LIN {X 0,Y 474.608,Z 139.367,A -85,B 0,C 180,E1 -7425.895,E2 -7425.895} C_VEL
LIN {X 0,Y 474.709,Z 139.486,A -85,B 0,C 180,E1 -7429.16,E2 -7429.16} C_VEL
LIN {X 0,Y 475.786,Z 146.089,A -85,B 0,C 180,E1 -7430.567,E2 -7430.567} C_VEL
LIN {X 0,Y 475.59,Z 156.694,A -85,B 0,C 180,E1 -7432.708,E2 -7432.708} C_VEL
LIN {X 0,Y 475.534,Z 159.268,A -85,B 0,C 180,E1 -7433.227,E2 -7433.227} C_VEL
LIN {X 0,Y 478.307,Z 173.098,A -85,B 0,C 180,E1 -7433.565,E2 -7433.565} C_VEL
LIN {X 0,Y 477.544,Z 266.711,A -85,B 0,C 180,E1 -7435.018,E2 -7435.018} C_VEL
LIN {X 0,Y 477.306,Z 280.071,A -85,B 0,C 180,E1 -7435.404,E2 -7435.404} C_VEL
LIN {X 0,Y 477.288,Z 280.718,A -85,B 0,C 180,E1 -7435.427,E2 -7435.427} C_VEL
LIN {X 0,Y 476.628,Z 286.343,A -85,B 0,C 180,E1 -7435.627,E2 -7435.627} C_VEL
LIN {X 0,Y 473.579,Z 295.359,A -85,B 0,C 180,E1 -7435.964,E2 -7435.964} C_VEL
LIN {X 0,Y 470.344,Z 304.06,A -85,B 0,C 180,E1 -7436.39,E2 -7436.39} C_VEL
LIN {X 0,Y 469.403,Z 309.194,A -85,B 0,C 180,E1 -7436.728,E2 -7436.728} C_VEL
LIN {X 0,Y 468.945,Z 319.732,A -85,B 0,C 180,E1 -7437.603,E2 -7437.603} C_VEL
LIN {X 0,Y 468.482,Z 329.529,A -85,B 0,C 180,E1 -7438.608,E2 -7438.608} C_VEL
LIN {X 0,Y 467.98,Z 338.944,A -85,B 0,C 180,E1 -7439.795,E2 -7439.795} C_VEL
LIN {X 0,Y 467.628,Z 346.312,A -85,B 0,C 180,E1 -7440.941,E2 -7440.941} C_VEL
LIN {X 0,Y 467.263,Z 352.96,A -85,B 0,C 180,E1 -7442.208,E2 -7442.208} C_VEL
LIN {X 0,Y 467.028,Z 358.937,A -85,B 0,C 180,E1 -7443.645,E2 -7443.645} C_VEL
LIN {X 0,Y 466.831,Z 363.471,A -85,B 0,C 180,E1 -7445.069,E2 -7445.069} C_VEL
LIN {X 0,Y 466.694,Z 367.163,A -85,B 0,C 180,E1 -7446.722,E2 -7446.722} C_VEL
LIN {X 0,Y 466.58,Z 368.845,A -85,B 0,C 180,E1 -7447.879,E2 -7447.879} C_VEL
LIN {X 0,Y 466.563,Z 369.776,A -85,B 0,C 180,E1 -7449.054,E2 -7449.054} C_VEL
LIN {X 0,Y 466.57,Z 369.919,A -85,B 0,C 180,E1 -7450.647,E2 -7450.647} C_VEL
LIN {X 0,Y 466.589,Z 369.328,A -85,B 0,C 180,E1 -7451.609,E2 -7451.609} C_VEL
LIN {X 0,Y 466.604,Z 368.392,A -85,B 0,C 180,E1 -7452.468,E2 -7452.468} C_VEL
LIN {X 0,Y 466.676,Z 366.991,A -85,B 0,C 180,E1 -7453.373,E2 -7453.373} C_VEL
LIN {X 0,Y 466.797,Z 364.598,A -85,B 0,C 180,E1 -7454.485,E2 -7454.485} C_VEL
LIN {X 0,Y 466.946,Z 359.956,A -85,B 0,C 180,E1 -7456.065,E2 -7456.065} C_VEL
LIN {X 0,Y 467.236,Z 353.669,A -85,B 0,C 180,E1 -7457.623,E2 -7457.623} C_VEL
LIN {X 0,Y 467.517,Z 346.823,A -85,B 0,C 180,E1 -7458.95,E2 -7458.95} C_VEL
LIN {X 0,Y 467.878,Z 338.315,A -85,B 0,C 180,E1 -7460.271,E2 -7460.271} C_VEL
LIN {X 0,Y 468.347,Z 329.513,A -85,B 0,C 180,E1 -7461.37,E2 -7461.37} C_VEL
LIN {X 0,Y 468.844,Z 318.706,A -85,B 0,C 180,E1 -7462.463,E2 -7462.463} C_VEL
LIN {X 0,Y 469.333,Z 307.899,A -85,B 0,C 180,E1 -7463.336,E2 -7463.336} C_VEL
LIN {X 0,Y 469.76,Z 295.801,A -85,B 0,C 180,E1 -7464.096,E2 -7464.096} C_VEL
LIN {X 0,Y 470.119,Z 283.179,A -85,B 0,C 180,E1 -7464.693,E2 -7464.693} C_VEL
LIN {X 0,Y 470.413,Z 270.759,A -85,B 0,C 180,E1 -7465.099,E2 -7465.099} C_VEL
LIN {X 0,Y 470.555,Z 255.199,A -85,B 0,C 180,E1 -7465.396,E2 -7465.396} C_VEL
LIN {X 0,Y 471.161,Z 173.344,A -85,B 0,C 180,E1 -7466.66,E2 -7466.66} C_VEL
LIN {X 0,Y 468.382,Z 159.359,A -85,B 0,C 180,E1 -7466.99,E2 -7466.99} C_VEL
LIN {X 0,Y 468.71,Z 147.809,A -85,B 0,C 180,E1 -7469.356,E2 -7469.356} C_VEL
LIN {X 0,Y 468.548,Z 144.722,A -85,B 0,C 180,E1 -7470,E2 -7470} C_VEL
LIN {X 0,Y 467.639,Z 140.235,A -85,B 0,C 180,E1 -7471.023,E2 -7471.023} C_VEL
LIN {X 0,Y 467.806,Z 140.215,A -85,B 0,C 180,E1 -7472.583,E2 -7472.583} C_VEL
LIN {X 0,Y 467.695,Z 140.229,A -85,B 0,C 180,E1 -7476.038,E2 -7476.038} C_VEL
LIN {X 0,Y 467.628,Z 140.231,A -85,B 0,C 180,E1 -7478.644,E2 -7478.644} C_VEL
LIN {X 0,Y 467.643,Z 140.232,A -85,B 0,C 180,E1 -7482.146,E2 -7482.146} C_VEL
LIN {X 0,Y 467.572,Z 140.246,A -85,B 0,C 180,E1 -7485.698,E2 -7485.698} C_VEL
LIN {X 0,Y 467.564,Z 140.239,A -85,B 0,C 180,E1 -7488.747,E2 -7488.747} C_VEL
LIN {X 0,Y 467.51,Z 140.247,A -85,B 0,C 180,E1 -7492.075,E2 -7492.075} C_VEL
LIN {X 0,Y 467.523,Z 140.245,A -85,B 0,C 180,E1 -7494.892,E2 -7494.892} C_VEL
LIN {X 0,Y 467.533,Z 140.246,A -85,B 0,C 180,E1 -7497.775,E2 -7497.775} C_VEL
LIN {X 0,Y 467.524,Z 140.248,A -85,B 0,C 180,E1 -7501.037,E2 -7501.037} C_VEL
LIN {X 0,Y 467.56,Z 140.239,A -85,B 0,C 180,E1 -7504.238,E2 -7504.238} C_VEL
LIN {X 0,Y 467.511,Z 140.253,A -85,B 0,C 180,E1 -7507.181,E2 -7507.181} C_VEL
LIN {X 0,Y 467.538,Z 140.242,A -85,B 0,C 180,E1 -7510.269,E2 -7510.269} C_VEL
LIN {X 0,Y 467.515,Z 140.247,A -85,B 0,C 180,E1 -7512.569,E2 -7512.569} C_VEL
LIN {X 0,Y 467.561,Z 140.246,A -85,B 0,C 180,E1 -7515.053,E2 -7515.053} C_VEL
LIN {X 0,Y 467.559,Z 140.246,A -85,B 0,C 180,E1 -7518.727,E2 -7518.727} C_VEL
LIN {X 0,Y 467.54,Z 140.242,A -85,B 0,C 180,E1 -7521.954,E2 -7521.954} C_VEL
LIN {X 0,Y 467.545,Z 140.243,A -85,B 0,C 180,E1 -7525.166,E2 -7525.166} C_VEL
LIN {X 0,Y 467.543,Z 140.245,A -85,B 0,C 180,E1 -7528.257,E2 -7528.257} C_VEL
LIN {X 0,Y 467.525,Z 140.244,A -85,B 0,C 180,E1 -7531.248,E2 -7531.248} C_VEL
LIN {X 0,Y 467.563,Z 140.246,A -85,B 0,C 180,E1 -7534.406,E2 -7534.406} C_VEL
LIN {X 0,Y 467.551,Z 140.242,A -85,B 0,C 180,E1 -7536.995,E2 -7536.995} C_VEL
LIN {X 0,Y 467.54,Z 140.243,A -85,B 0,C 180,E1 -7539.774,E2 -7539.774} C_VEL
LIN {X 0,Y 467.554,Z 140.245,A -85,B 0,C 180,E1 -7542.505,E2 -7542.505} C_VEL
LIN {X 0,Y 467.564,Z 140.239,A -85,B 0,C 180,E1 -7545.196,E2 -7545.196} C_VEL
LIN {X 0,Y 467.652,Z 140.232,A -85,B 0,C 180,E1 -7547.855,E2 -7547.855} C_VEL
LIN {X 0,Y 467.633,Z 140.231,A -85,B 0,C 180,E1 -7551.357,E2 -7551.357} C_VEL
LIN {X 0,Y 467.704,Z 140.229,A -85,B 0,C 180,E1 -7553.963,E2 -7553.963} C_VEL
LIN {X 0,Y 467.815,Z 140.21,A -85,B 0,C 180,E1 -7557.417,E2 -7557.417} C_VEL
LIN {X 0,Y 467.853,Z 140.208,A -85,B 0,C 180,E1 -7560,E2 -7560} C_VEL
LIN {X 0,Y 467.815,Z 140.208,A -85,B 0,C 180,E1 -7562.584,E2 -7562.584} C_VEL
LIN {X 0,Y 467.698,Z 140.225,A -85,B 0,C 180,E1 -7566.038,E2 -7566.038} C_VEL
LIN {X 0,Y 467.64,Z 140.229,A -85,B 0,C 180,E1 -7568.644,E2 -7568.644} C_VEL
LIN {X 0,Y 467.662,Z 140.228,A -85,B 0,C 180,E1 -7572.146,E2 -7572.146} C_VEL
LIN {X 0,Y 467.618,Z 140.237,A -85,B 0,C 180,E1 -7575.696,E2 -7575.696} C_VEL
LIN {X 0,Y 467.62,Z 140.239,A -85,B 0,C 180,E1 -7579.308,E2 -7579.308} C_VEL
LIN {X 0,Y 467.529,Z 140.243,A -85,B 0,C 180,E1 -7582.075,E2 -7582.075} C_VEL
LIN {X 0,Y 467.56,Z 140.243,A -85,B 0,C 180,E1 -7584.89,E2 -7584.89} C_VEL
LIN {X 0,Y 467.548,Z 140.242,A -85,B 0,C 180,E1 -7587.774,E2 -7587.774} C_VEL
LIN {X 0,Y 467.542,Z 140.249,A -85,B 0,C 180,E1 -7591.038,E2 -7591.038} C_VEL
LIN {X 0,Y 467.581,Z 140.237,A -85,B 0,C 180,E1 -7594.24,E2 -7594.24} C_VEL
LIN {X 0,Y 467.547,Z 140.245,A -85,B 0,C 180,E1 -7597.185,E2 -7597.185} C_VEL
LIN {X 0,Y 467.562,Z 140.241,A -85,B 0,C 180,E1 -7600.267,E2 -7600.267} C_VEL
LIN {X 0,Y 467.549,Z 140.241,A -85,B 0,C 180,E1 -7603.746,E2 -7603.746} C_VEL
LIN {X 0,Y 467.549,Z 140.243,A -85,B 0,C 180,E1 -7606.254,E2 -7606.254} C_VEL
LIN {X 0,Y 467.561,Z 140.239,A -85,B 0,C 180,E1 -7609.733,E2 -7609.733} C_VEL
LIN {X 0,Y 467.546,Z 140.245,A -85,B 0,C 180,E1 -7612.815,E2 -7612.815} C_VEL
LIN {X 0,Y 467.58,Z 140.238,A -85,B 0,C 180,E1 -7615.76,E2 -7615.76} C_VEL
LIN {X 0,Y 467.569,Z 140.242,A -85,B 0,C 180,E1 -7618.956,E2 -7618.956} C_VEL
LIN {X 0,Y 467.549,Z 140.25,A -85,B 0,C 180,E1 -7622.226,E2 -7622.226} C_VEL
LIN {X 0,Y 467.586,Z 140.323,A -85,B 0,C 180,E1 -7624.069,E2 -7624.069} C_VEL
LIN {X 0,Y 469.75,Z 151.558,A -85,B 0,C 180,E1 -7626.174,E2 -7626.174} C_VEL
LIN {X 0,Y 469.254,Z 166.324,A -85,B 0,C 180,E1 -7628.746,E2 -7628.746} C_VEL
LIN {X 0,Y 468.414,Z 185.761,A -85,B 0,C 180,E1 -7632.086,E2 -7632.086} C_VEL
LIN {X 0,Y 468.271,Z 191.496,A -85,B 0,C 180,E1 -7633.045,E2 -7633.045} C_VEL
LIN {X 0,Y 471.064,Z 211.651,A -85,B 0,C 180,E1 -7633.456,E2 -7633.456} C_VEL
LIN {X 0,Y 470.402,Z 300.211,A -85,B 0,C 180,E1 -7634.843,E2 -7634.843} C_VEL
LIN {X 0,Y 470.047,Z 313.325,A -85,B 0,C 180,E1 -7635.219,E2 -7635.219} C_VEL
LIN {X 0,Y 469.617,Z 324.856,A -85,B 0,C 180,E1 -7635.704,E2 -7635.704} C_VEL
LIN {X 0,Y 469.114,Z 336.418,A -85,B 0,C 180,E1 -7636.352,E2 -7636.352} C_VEL
LIN {X 0,Y 468.642,Z 348.04,A -85,B 0,C 180,E1 -7637.201,E2 -7637.201} C_VEL
LIN {X 0,Y 468.175,Z 358.889,A -85,B 0,C 180,E1 -7638.198,E2 -7638.198} C_VEL
LIN {X 0,Y 467.738,Z 367.56,A -85,B 0,C 180,E1 -7639.174,E2 -7639.174} C_VEL
LIN {X 0,Y 467.413,Z 375.553,A -85,B 0,C 180,E1 -7640.261,E2 -7640.261} C_VEL
LIN {X 0,Y 467.087,Z 383.366,A -85,B 0,C 180,E1 -7641.564,E2 -7641.564} C_VEL
LIN {X 0,Y 466.831,Z 390.534,A -85,B 0,C 180,E1 -7643.082,E2 -7643.082} C_VEL
LIN {X 0,Y 466.73,Z 395.31,A -85,B 0,C 180,E1 -7644.383,E2 -7644.383} C_VEL
LIN {X 0,Y 466.646,Z 398.958,A -85,B 0,C 180,E1 -7645.681,E2 -7645.681} C_VEL
LIN {X 0,Y 466.69,Z 400.845,A -85,B 0,C 180,E1 -7646.546,E2 -7646.546} C_VEL
LIN {X 0,Y 466.662,Z 402.259,A -85,B 0,C 180,E1 -7647.41,E2 -7647.41} C_VEL
LIN {X 0,Y 466.623,Z 403.879,A -85,B 0,C 180,E1 -7649.137,E2 -7649.137} C_VEL
LIN {X 0,Y 466.605,Z 404.104,A -85,B 0,C 180,E1 -7650,E2 -7650} C_VEL
LIN {X 0,Y 466.623,Z 403.896,A -85,B 0,C 180,E1 -7650.863,E2 -7650.863} C_VEL
LIN {X 0,Y 466.662,Z 402.295,A -85,B 0,C 180,E1 -7652.589,E2 -7652.589} C_VEL
LIN {X 0,Y 466.689,Z 400.901,A -85,B 0,C 180,E1 -7653.453,E2 -7653.453} C_VEL
LIN {X 0,Y 466.687,Z 397.963,A -85,B 0,C 180,E1 -7654.751,E2 -7654.751} C_VEL
LIN {X 0,Y 466.725,Z 393.99,A -85,B 0,C 180,E1 -7656.05,E2 -7656.05} C_VEL
LIN {X 0,Y 466.938,Z 387.896,A -85,B 0,C 180,E1 -7657.568,E2 -7657.568} C_VEL
LIN {X 0,Y 467.178,Z 381.231,A -85,B 0,C 180,E1 -7658.87,E2 -7658.87} C_VEL
LIN {X 0,Y 467.5,Z 372.967,A -85,B 0,C 180,E1 -7660.174,E2 -7660.174} C_VEL
LIN {X 0,Y 467.977,Z 364.522,A -85,B 0,C 180,E1 -7661.258,E2 -7661.258} C_VEL
LIN {X 0,Y 468.416,Z 354.6,A -85,B 0,C 180,E1 -7662.299,E2 -7662.299} C_VEL
LIN {X 0,Y 468.902,Z 343.815,A -85,B 0,C 180,E1 -7663.213,E2 -7663.213} C_VEL
LIN {X 0,Y 469.449,Z 332.569,A -85,B 0,C 180,E1 -7663.969,E2 -7663.969} C_VEL
LIN {X 0,Y 469.961,Z 321.173,A -85,B 0,C 180,E1 -7664.562,E2 -7664.562} C_VEL
LIN {X 0,Y 470.38,Z 308.209,A -85,B 0,C 180,E1 -7665.046,E2 -7665.046} C_VEL
LIN {X 0,Y 470.76,Z 294.419,A -85,B 0,C 180,E1 -7665.366,E2 -7665.366} C_VEL
LIN {X 0,Y 471.211,Z 209.62,A -85,B 0,C 180,E1 -7666.69,E2 -7666.69} C_VEL
LIN {X 0,Y 468.299,Z 190.956,A -85,B 0,C 180,E1 -7667.111,E2 -7667.111} C_VEL
LIN {X 0,Y 468.996,Z 173.231,A -85,B 0,C 180,E1 -7670.161,E2 -7670.161} C_VEL
LIN {X 0,Y 469.879,Z 154.997,A -85,B 0,C 180,E1 -7673.351,E2 -7673.351} C_VEL
LIN {X 0,Y 469.707,Z 150.782,A -85,B 0,C 180,E1 -7674.116,E2 -7674.116} C_VEL
LIN {X 0,Y 467.582,Z 140.244,A -85,B 0,C 180,E1 -7676.171,E2 -7676.171} C_VEL
LIN {X 0,Y 467.553,Z 140.251,A -85,B 0,C 180,E1 -7679.328,E2 -7679.328} C_VEL
LIN {X 0,Y 467.58,Z 140.242,A -85,B 0,C 180,E1 -7681.74,E2 -7681.74} C_VEL
LIN {X 0,Y 467.556,Z 140.239,A -85,B 0,C 180,E1 -7684.833,E2 -7684.833} C_VEL
LIN {X 0,Y 467.554,Z 140.243,A -85,B 0,C 180,E1 -7688.046,E2 -7688.046} C_VEL
LIN {X 0,Y 467.562,Z 140.241,A -85,B 0,C 180,E1 -7691.274,E2 -7691.274} C_VEL
LIN {X 0,Y 467.566,Z 140.244,A -85,B 0,C 180,E1 -7694.948,E2 -7694.948} C_VEL
LIN {X 0,Y 467.556,Z 140.244,A -85,B 0,C 180,E1 -7698.594,E2 -7698.594} C_VEL
LIN {X 0,Y 467.537,Z 140.241,A -85,B 0,C 180,E1 -7701.952,E2 -7701.952} C_VEL
LIN {X 0,Y 467.54,Z 140.243,A -85,B 0,C 180,E1 -7705.165,E2 -7705.165} C_VEL
LIN {X 0,Y 467.544,Z 140.245,A -85,B 0,C 180,E1 -7708.257,E2 -7708.257} C_VEL
LIN {X 0,Y 467.527,Z 140.244,A -85,B 0,C 180,E1 -7711.247,E2 -7711.247} C_VEL
LIN {X 0,Y 467.564,Z 140.242,A -85,B 0,C 180,E1 -7714.405,E2 -7714.405} C_VEL
LIN {X 0,Y 467.552,Z 140.237,A -85,B 0,C 180,E1 -7716.994,E2 -7716.994} C_VEL
LIN {X 0,Y 467.537,Z 140.244,A -85,B 0,C 180,E1 -7719.773,E2 -7719.773} C_VEL
LIN {X 0,Y 467.555,Z 140.243,A -85,B 0,C 180,E1 -7722.504,E2 -7722.504} C_VEL
LIN {X 0,Y 467.592,Z 140.236,A -85,B 0,C 180,E1 -7725.196,E2 -7725.196} C_VEL
LIN {X 0,Y 467.651,Z 140.228,A -85,B 0,C 180,E1 -7727.854,E2 -7727.854} C_VEL
LIN {X 0,Y 467.658,Z 140.226,A -85,B 0,C 180,E1 -7731.356,E2 -7731.356} C_VEL
LIN {X 0,Y 467.706,Z 140.227,A -85,B 0,C 180,E1 -7733.962,E2 -7733.962} C_VEL
LIN {X 0,Y 467.816,Z 140.205,A -85,B 0,C 180,E1 -7737.416,E2 -7737.416} C_VEL
LIN {X 0,Y 467.855,Z 140.203,A -85,B 0,C 180,E1 -7740,E2 -7740} C_VEL
LIN {X 0,Y 467.852,Z 140.202,A -85,B 0,C 180,E1 -7742.582,E2 -7742.582} C_VEL
LIN {X 0,Y 467.715,Z 140.218,A -85,B 0,C 180,E1 -7746.037,E2 -7746.037} C_VEL
LIN {X 0,Y 467.669,Z 140.227,A -85,B 0,C 180,E1 -7748.642,E2 -7748.642} C_VEL
LIN {X 0,Y 467.658,Z 140.228,A -85,B 0,C 180,E1 -7752.145,E2 -7752.145} C_VEL
LIN {X 0,Y 467.64,Z 140.232,A -85,B 0,C 180,E1 -7755.694,E2 -7755.694} C_VEL
LIN {X 0,Y 467.622,Z 140.237,A -85,B 0,C 180,E1 -7759.307,E2 -7759.307} C_VEL
LIN {X 0,Y 467.535,Z 140.24,A -85,B 0,C 180,E1 -7762.073,E2 -7762.073} C_VEL
LIN {X 0,Y 467.579,Z 140.243,A -85,B 0,C 180,E1 -7764.888,E2 -7764.888} C_VEL
LIN {X 0,Y 467.616,Z 140.233,A -85,B 0,C 180,E1 -7767.769,E2 -7767.769} C_VEL
LIN {X 0,Y 467.567,Z 140.243,A -85,B 0,C 180,E1 -7771.044,E2 -7771.044} C_VEL
LIN {X 0,Y 467.576,Z 140.243,A -85,B 0,C 180,E1 -7774.24,E2 -7774.24} C_VEL
LIN {X 0,Y 467.547,Z 140.246,A -85,B 0,C 180,E1 -7777.186,E2 -7777.186} C_VEL
LIN {X 0,Y 467.576,Z 140.247,A -85,B 0,C 180,E1 -7780.264,E2 -7780.264} C_VEL
LIN {X 0,Y 467.585,Z 140.247,A -85,B 0,C 180,E1 -7782.566,E2 -7782.566} C_VEL
LIN {X 0,Y 467.569,Z 140.243,A -85,B 0,C 180,E1 -7785.053,E2 -7785.053} C_VEL
LIN {X 0,Y 467.619,Z 140.24,A -85,B 0,C 180,E1 -7788.601,E2 -7788.601} C_VEL
LIN {X 0,Y 467.678,Z 140.464,A -85,B 0,C 180,E1 -7788.974,E2 -7788.974} C_VEL
LIN {X 0,Y 468.839,Z 147.182,A -85,B 0,C 180,E1 -7790.425,E2 -7790.425} C_VEL
LIN {X 0,Y 468.68,Z 156.803,A -85,B 0,C 180,E1 -7792.4,E2 -7792.4} C_VEL
LIN {X 0,Y 468.599,Z 159.522,A -85,B 0,C 180,E1 -7792.953,E2 -7792.953} C_VEL
LIN {X 0,Y 471.593,Z 174.295,A -85,B 0,C 180,E1 -7793.322,E2 -7793.322} C_VEL
LIN {X 0,Y 470.755,Z 267.078,A -85,B 0,C 180,E1 -7794.783,E2 -7794.783} C_VEL
LIN {X 0,Y 470.484,Z 280.282,A -85,B 0,C 180,E1 -7795.17,E2 -7795.17} C_VEL
LIN {X 0,Y 470.105,Z 292.719,A -85,B 0,C 180,E1 -7795.707,E2 -7795.707} C_VEL
LIN {X 0,Y 469.661,Z 304.233,A -85,B 0,C 180,E1 -7796.381,E2 -7796.381} C_VEL
LIN {X 0,Y 469.403,Z 309.194,A -85,B 0,C 180,E1 -7796.728,E2 -7796.728} C_VEL
LIN {X 0,Y 468.5,Z 314.228,A -85,B 0,C 180,E1 -7797.098,E2 -7797.098} C_VEL
LIN {X 0,Y 465.345,Z 322.192,A -85,B 0,C 180,E1 -7797.719,E2 -7797.719} C_VEL
LIN {X 0,Y 462.2,Z 329.652,A -85,B 0,C 180,E1 -7798.42,E2 -7798.42} C_VEL
LIN {X 0,Y 461.313,Z 333.878,A -85,B 0,C 180,E1 -7798.91,E2 -7798.91} C_VEL
LIN {X 0,Y 460.81,Z 342.638,A -85,B 0,C 180,E1 -7800.135,E2 -7800.135} C_VEL
LIN {X 0,Y 460.366,Z 350.469,A -85,B 0,C 180,E1 -7801.506,E2 -7801.506} C_VEL
LIN {X 0,Y 460.132,Z 356.099,A -85,B 0,C 180,E1 -7802.728,E2 -7802.728} C_VEL
LIN {X 0,Y 459.891,Z 361.081,A -85,B 0,C 180,E1 -7804.082,E2 -7804.082} C_VEL
LIN {X 0,Y 459.697,Z 365.338,A -85,B 0,C 180,E1 -7805.62,E2 -7805.62} C_VEL
LIN {X 0,Y 459.609,Z 367.294,A -85,B 0,C 180,E1 -7806.573,E2 -7806.573} C_VEL
LIN {X 0,Y 459.508,Z 368.717,A -85,B 0,C 180,E1 -7807.52,E2 -7807.52} C_VEL
LIN {X 0,Y 459.476,Z 369.978,A -85,B 0,C 180,E1 -7808.912,E2 -7808.912} C_VEL
LIN {X 0,Y 459.488,Z 370.236,A -85,B 0,C 180,E1 -7810.336,E2 -7810.336} C_VEL
LIN {X 0,Y 459.489,Z 369.698,A -85,B 0,C 180,E1 -7811.495,E2 -7811.495} C_VEL
LIN {X 0,Y 459.571,Z 367.742,A -85,B 0,C 180,E1 -7813.109,E2 -7813.109} C_VEL
LIN {X 0,Y 459.708,Z 365.199,A -85,B 0,C 180,E1 -7814.393,E2 -7814.393} C_VEL
LIN {X 0,Y 459.842,Z 361.165,A -85,B 0,C 180,E1 -7815.846,E2 -7815.846} C_VEL
LIN {X 0,Y 460.047,Z 356.182,A -85,B 0,C 180,E1 -7817.202,E2 -7817.202} C_VEL
LIN {X 0,Y 460.306,Z 349.905,A -85,B 0,C 180,E1 -7818.552,E2 -7818.552} C_VEL
LIN {X 0,Y 460.712,Z 342.057,A -85,B 0,C 180,E1 -7819.896,E2 -7819.896} C_VEL
LIN {X 0,Y 461.124,Z 334.025,A -85,B 0,C 180,E1 -7821.013,E2 -7821.013} C_VEL
LIN {X 0,Y 461.622,Z 324.229,A -85,B 0,C 180,E1 -7822.125,E2 -7822.125} C_VEL
LIN {X 0,Y 462.202,Z 313.304,A -85,B 0,C 180,E1 -7823.123,E2 -7823.123} C_VEL
LIN {X 0,Y 462.644,Z 302.651,A -85,B 0,C 180,E1 -7823.896,E2 -7823.896} C_VEL
LIN {X 0,Y 463.035,Z 289.889,A -85,B 0,C 180,E1 -7824.611,E2 -7824.611} C_VEL
LIN {X 0,Y 463.383,Z 276.985,A -85,B 0,C 180,E1 -7825.133,E2 -7825.133} C_VEL
LIN {X 0,Y 463.63,Z 264.209,A -85,B 0,C 180,E1 -7825.463,E2 -7825.463} C_VEL
LIN {X 0,Y 464.368,Z 174.501,A -85,B 0,C 180,E1 -7826.877,E2 -7826.877} C_VEL
LIN {X 0,Y 461.426,Z 159.593,A -85,B 0,C 180,E1 -7827.233,E2 -7827.233} C_VEL
LIN {X 0,Y 461.74,Z 148.329,A -85,B 0,C 180,E1 -7829.564,E2 -7829.564} C_VEL
LIN {X 0,Y 461.215,Z 144.287,A -85,B 0,C 180,E1 -7830.437,E2 -7830.437} C_VEL
LIN {X 0,Y 460.625,Z 141.109,A -85,B 0,C 180,E1 -7831.148,E2 -7831.148} C_VEL
LIN {X 0,Y 460.75,Z 141.094,A -85,B 0,C 180,E1 -7832.623,E2 -7832.623} C_VEL
LIN {X 0,Y 460.661,Z 141.104,A -85,B 0,C 180,E1 -7836.131,E2 -7836.131} C_VEL
LIN {X 0,Y 460.583,Z 141.108,A -85,B 0,C 180,E1 -7838.777,E2 -7838.777} C_VEL
LIN {X 0,Y 460.593,Z 141.108,A -85,B 0,C 180,E1 -7842.435,E2 -7842.435} C_VEL
LIN {X 0,Y 460.521,Z 141.12,A -85,B 0,C 180,E1 -7845.965,E2 -7845.965} C_VEL
LIN {X 0,Y 460.522,Z 141.117,A -85,B 0,C 180,E1 -7848.885,E2 -7848.885} C_VEL
LIN {X 0,Y 460.484,Z 141.121,A -85,B 0,C 180,E1 -7852.43,E2 -7852.43} C_VEL
LIN {X 0,Y 460.517,Z 141.12,A -85,B 0,C 180,E1 -7855.79,E2 -7855.79} C_VEL
LIN {X 0,Y 460.491,Z 141.12,A -85,B 0,C 180,E1 -7858.237,E2 -7858.237} C_VEL
LIN {X 0,Y 460.492,Z 141.128,A -85,B 0,C 180,E1 -7861.278,E2 -7861.278} C_VEL
LIN {X 0,Y 460.507,Z 141.118,A -85,B 0,C 180,E1 -7864.502,E2 -7864.502} C_VEL
LIN {X 0,Y 460.478,Z 141.124,A -85,B 0,C 180,E1 -7867.626,E2 -7867.626} C_VEL
LIN {X 0,Y 460.505,Z 141.126,A -85,B 0,C 180,E1 -7871.015,E2 -7871.015} C_VEL
LIN {X 0,Y 460.508,Z 141.121,A -85,B 0,C 180,E1 -7874.59,E2 -7874.59} C_VEL
LIN {X 0,Y 460.472,Z 141.122,A -85,B 0,C 180,E1 -7877.814,E2 -7877.814} C_VEL
LIN {X 0,Y 460.509,Z 141.118,A -85,B 0,C 180,E1 -7880.136,E2 -7880.136} C_VEL
LIN {X 0,Y 460.46,Z 141.124,A -85,B 0,C 180,E1 -7883.47,E2 -7883.47} C_VEL
LIN {X 0,Y 460.501,Z 141.127,A -85,B 0,C 180,E1 -7886.673,E2 -7886.673} C_VEL
LIN {X 0,Y 460.479,Z 141.122,A -85,B 0,C 180,E1 -7889.758,E2 -7889.758} C_VEL
LIN {X 0,Y 460.485,Z 141.125,A -85,B 0,C 180,E1 -7892.751,E2 -7892.751} C_VEL
LIN {X 0,Y 460.498,Z 141.119,A -85,B 0,C 180,E1 -7895.666,E2 -7895.666} C_VEL
LIN {X 0,Y 460.512,Z 141.122,A -85,B 0,C 180,E1 -7898.583,E2 -7898.583} C_VEL
LIN {X 0,Y 460.529,Z 141.115,A -85,B 0,C 180,E1 -7901.309,E2 -7901.309} C_VEL
LIN {X 0,Y 460.523,Z 141.121,A -85,B 0,C 180,E1 -7904.057,E2 -7904.057} C_VEL
LIN {X 0,Y 460.607,Z 141.108,A -85,B 0,C 180,E1 -7907.666,E2 -7907.666} C_VEL
LIN {X 0,Y 460.589,Z 141.108,A -85,B 0,C 180,E1 -7911.224,E2 -7911.224} C_VEL
LIN {X 0,Y 460.67,Z 141.104,A -85,B 0,C 180,E1 -7913.87,E2 -7913.87} C_VEL
LIN {X 0,Y 460.759,Z 141.088,A -85,B 0,C 180,E1 -7917.378,E2 -7917.378} C_VEL
LIN {X 0,Y 460.823,Z 141.084,A -85,B 0,C 180,E1 -7920,E2 -7920} C_VEL
LIN {X 0,Y 460.759,Z 141.087,A -85,B 0,C 180,E1 -7922.623,E2 -7922.623} C_VEL
LIN {X 0,Y 460.665,Z 141.101,A -85,B 0,C 180,E1 -7926.131,E2 -7926.131} C_VEL
LIN {X 0,Y 460.595,Z 141.107,A -85,B 0,C 180,E1 -7928.777,E2 -7928.777} C_VEL
LIN {X 0,Y 460.615,Z 141.105,A -85,B 0,C 180,E1 -7932.334,E2 -7932.334} C_VEL
LIN {X 0,Y 460.562,Z 141.113,A -85,B 0,C 180,E1 -7935.979,E2 -7935.979} C_VEL
LIN {X 0,Y 460.565,Z 141.115,A -85,B 0,C 180,E1 -7939.616,E2 -7939.616} C_VEL
LIN {X 0,Y 460.507,Z 141.118,A -85,B 0,C 180,E1 -7942.429,E2 -7942.429} C_VEL
LIN {X 0,Y 460.538,Z 141.115,A -85,B 0,C 180,E1 -7945.793,E2 -7945.793} C_VEL
LIN {X 0,Y 460.519,Z 141.123,A -85,B 0,C 180,E1 -7949.233,E2 -7949.233} C_VEL
LIN {X 0,Y 460.519,Z 141.117,A -85,B 0,C 180,E1 -7952.286,E2 -7952.286} C_VEL
LIN {X 0,Y 460.511,Z 141.119,A -85,B 0,C 180,E1 -7955.446,E2 -7955.446} C_VEL
LIN {X 0,Y 460.534,Z 141.122,A -85,B 0,C 180,E1 -7958.895,E2 -7958.895} C_VEL
LIN {X 0,Y 460.506,Z 141.118,A -85,B 0,C 180,E1 -7961.598,E2 -7961.598} C_VEL
LIN {X 0,Y 460.515,Z 141.123,A -85,B 0,C 180,E1 -7964.589,E2 -7964.589} C_VEL
LIN {X 0,Y 460.479,Z 141.122,A -85,B 0,C 180,E1 -7967.813,E2 -7967.813} C_VEL
LIN {X 0,Y 460.517,Z 141.119,A -85,B 0,C 180,E1 -7970.135,E2 -7970.135} C_VEL
LIN {X 0,Y 460.476,Z 141.122,A -85,B 0,C 180,E1 -7973.47,E2 -7973.47} C_VEL
LIN {X 0,Y 460.52,Z 141.121,A -85,B 0,C 180,E1 -7976.674,E2 -7976.674} C_VEL
LIN {X 0,Y 460.508,Z 141.122,A -85,B 0,C 180,E1 -7979.759,E2 -7979.759} C_VEL
LIN {X 0,Y 460.497,Z 141.128,A -85,B 0,C 180,E1 -7982.751,E2 -7982.751} C_VEL
LIN {X 0,Y 460.56,Z 141.302,A -85,B 0,C 180,E1 -7983.898,E2 -7983.898} C_VEL
LIN {X 0,Y 462.74,Z 152.477,A -85,B 0,C 180,E1 -7986.029,E2 -7986.029} C_VEL
LIN {X 0,Y 462.383,Z 163.581,A -85,B 0,C 180,E1 -7987.999,E2 -7987.999} C_VEL
LIN {X 0,Y 461.507,Z 184.093,A -85,B 0,C 180,E1 -7991.579,E2 -7991.579} C_VEL
LIN {X 0,Y 461.269,Z 190.976,A -85,B 0,C 180,E1 -7992.773,E2 -7992.773} C_VEL
LIN {X 0,Y 464.218,Z 212.178,A -85,B 0,C 180,E1 -7993.236,E2 -7993.236} C_VEL
LIN {X 0,Y 463.508,Z 300.324,A -85,B 0,C 180,E1 -7994.64,E2 -7994.64} C_VEL
LIN {X 0,Y 463.14,Z 313.314,A -85,B 0,C 180,E1 -7995.022,E2 -7995.022} C_VEL
LIN {X 0,Y 462.683,Z 325.349,A -85,B 0,C 180,E1 -7995.541,E2 -7995.541} C_VEL
LIN {X 0,Y 462.096,Z 337.516,A -85,B 0,C 180,E1 -7996.252,E2 -7996.252} C_VEL
LIN {X 0,Y 461.6,Z 349.544,A -85,B 0,C 180,E1 -7997.172,E2 -7997.172} C_VEL
LIN {X 0,Y 461.138,Z 359.527,A -85,B 0,C 180,E1 -7998.126,E2 -7998.126} C_VEL
LIN {X 0,Y 460.619,Z 368.89,A -85,B 0,C 180,E1 -7999.227,E2 -7999.227} C_VEL
LIN {X 0,Y 460.194,Z 377.959,A -85,B 0,C 180,E1 -8000.551,E2 -8000.551} C_VEL
LIN {X 0,Y 459.921,Z 385.266,A -85,B 0,C 180,E1 -8001.874,E2 -8001.874} C_VEL
LIN {X 0,Y 459.722,Z 391.482,A -85,B 0,C 180,E1 -8003.294,E2 -8003.294} C_VEL
LIN {X 0,Y 459.641,Z 396.334,A -85,B 0,C 180,E1 -8004.736,E2 -8004.736} C_VEL
LIN {X 0,Y 459.563,Z 398.657,A -85,B 0,C 180,E1 -8005.614,E2 -8005.614} C_VEL
LIN {X 0,Y 459.586,Z 400.551,A -85,B 0,C 180,E1 -8006.493,E2 -8006.493} C_VEL
LIN {X 0,Y 459.585,Z 401.979,A -85,B 0,C 180,E1 -8007.37,E2 -8007.37} C_VEL
LIN {X 0,Y 459.555,Z 403.612,A -85,B 0,C 180,E1 -8009.124,E2 -8009.124} C_VEL
LIN {X 0,Y 459.536,Z 403.844,A -85,B 0,C 180,E1 -8010,E2 -8010} C_VEL
LIN {X 0,Y 459.526,Z 403.645,A -85,B 0,C 180,E1 -8010.876,E2 -8010.876} C_VEL
LIN {X 0,Y 459.585,Z 402.056,A -85,B 0,C 180,E1 -8012.629,E2 -8012.629} C_VEL
LIN {X 0,Y 459.584,Z 400.668,A -85,B 0,C 180,E1 -8013.507,E2 -8013.507} C_VEL
LIN {X 0,Y 459.614,Z 397.74,A -85,B 0,C 180,E1 -8014.824,E2 -8014.824} C_VEL
LIN {X 0,Y 459.636,Z 393.093,A -85,B 0,C 180,E1 -8016.342,E2 -8016.342} C_VEL
LIN {X 0,Y 459.867,Z 387.705,A -85,B 0,C 180,E1 -8017.685,E2 -8017.685} C_VEL
LIN {X 0,Y 460.108,Z 381.054,A -85,B 0,C 180,E1 -8019.008,E2 -8019.008} C_VEL
LIN {X 0,Y 460.462,Z 372.807,A -85,B 0,C 180,E1 -8020.331,E2 -8020.331} C_VEL
LIN {X 0,Y 460.983,Z 364.385,A -85,B 0,C 180,E1 -8021.431,E2 -8021.431} C_VEL
LIN {X 0,Y 461.448,Z 354.703,A -85,B 0,C 180,E1 -8022.468,E2 -8022.468} C_VEL
LIN {X 0,Y 461.977,Z 343.75,A -85,B 0,C 180,E1 -8023.415,E2 -8023.415} C_VEL
LIN {X 0,Y 462.566,Z 332.553,A -85,B 0,C 180,E1 -8024.181,E2 -8024.181} C_VEL
LIN {X 0,Y 463.098,Z 321.231,A -85,B 0,C 180,E1 -8024.782,E2 -8024.782} C_VEL
LIN {X 0,Y 463.55,Z 308.46,A -85,B 0,C 180,E1 -8025.273,E2 -8025.273} C_VEL
LIN {X 0,Y 463.937,Z 295.007,A -85,B 0,C 180,E1 -8025.598,E2 -8025.598} C_VEL
LIN {X 0,Y 464.435,Z 210.149,A -85,B 0,C 180,E1 -8026.946,E2 -8026.946} C_VEL
LIN {X 0,Y 461.365,Z 190.618,A -85,B 0,C 180,E1 -8027.407,E2 -8027.407} C_VEL
LIN {X 0,Y 462.04,Z 174.427,A -85,B 0,C 180,E1 -8030.246,E2 -8030.246} C_VEL
LIN {X 0,Y 462.964,Z 156.195,A -85,B 0,C 180,E1 -8033.484,E2 -8033.484} C_VEL
LIN {X 0,Y 462.699,Z 151.758,A -85,B 0,C 180,E1 -8034.307,E2 -8034.307} C_VEL
LIN {X 0,Y 460.517,Z 141.124,A -85,B 0,C 180,E1 -8036.421,E2 -8036.421} C_VEL
LIN {X 0,Y 460.519,Z 141.126,A -85,B 0,C 180,E1 -8039.555,E2 -8039.555} C_VEL
LIN {X 0,Y 460.528,Z 141.118,A -85,B 0,C 180,E1 -8042.285,E2 -8042.285} C_VEL
LIN {X 0,Y 460.507,Z 141.124,A -85,B 0,C 180,E1 -8045.446,E2 -8045.446} C_VEL
LIN {X 0,Y 460.496,Z 141.124,A -85,B 0,C 180,E1 -8048.89,E2 -8048.89} C_VEL
LIN {X 0,Y 460.504,Z 141.122,A -85,B 0,C 180,E1 -8051.598,E2 -8051.598} C_VEL
LIN {X 0,Y 460.512,Z 141.119,A -85,B 0,C 180,E1 -8054.589,E2 -8054.589} C_VEL
LIN {X 0,Y 460.475,Z 141.124,A -85,B 0,C 180,E1 -8057.813,E2 -8057.813} C_VEL
LIN {X 0,Y 460.496,Z 141.12,A -85,B 0,C 180,E1 -8060.133,E2 -8060.133} C_VEL
LIN {X 0,Y 460.457,Z 141.127,A -85,B 0,C 180,E1 -8063.468,E2 -8063.468} C_VEL
LIN {X 0,Y 460.5,Z 141.123,A -85,B 0,C 180,E1 -8066.672,E2 -8066.672} C_VEL
LIN {X 0,Y 460.48,Z 141.119,A -85,B 0,C 180,E1 -8069.757,E2 -8069.757} C_VEL
LIN {X 0,Y 460.486,Z 141.121,A -85,B 0,C 180,E1 -8072.75,E2 -8072.75} C_VEL
LIN {X 0,Y 460.513,Z 141.118,A -85,B 0,C 180,E1 -8075.666,E2 -8075.666} C_VEL
LIN {X 0,Y 460.512,Z 141.122,A -85,B 0,C 180,E1 -8078.582,E2 -8078.582} C_VEL
LIN {X 0,Y 460.528,Z 141.113,A -85,B 0,C 180,E1 -8081.308,E2 -8081.308} C_VEL
LIN {X 0,Y 460.57,Z 141.116,A -85,B 0,C 180,E1 -8084.057,E2 -8084.057} C_VEL
LIN {X 0,Y 460.606,Z 141.103,A -85,B 0,C 180,E1 -8087.665,E2 -8087.665} C_VEL
LIN {X 0,Y 460.607,Z 141.104,A -85,B 0,C 180,E1 -8091.223,E2 -8091.223} C_VEL
LIN {X 0,Y 460.672,Z 141.104,A -85,B 0,C 180,E1 -8093.869,E2 -8093.869} C_VEL
LIN {X 0,Y 460.76,Z 141.083,A -85,B 0,C 180,E1 -8097.377,E2 -8097.377} C_VEL
LIN {X 0,Y 460.824,Z 141.079,A -85,B 0,C 180,E1 -8100,E2 -8100} C_VEL
LIN {X 0,Y 460.792,Z 141.081,A -85,B 0,C 180,E1 -8102.622,E2 -8102.622} C_VEL
LIN {X 0,Y 460.68,Z 141.094,A -85,B 0,C 180,E1 -8106.13,E2 -8106.13} C_VEL
LIN {X 0,Y 460.62,Z 141.106,A -85,B 0,C 180,E1 -8108.776,E2 -8108.776} C_VEL
LIN {X 0,Y 460.616,Z 141.106,A -85,B 0,C 180,E1 -8112.444,E2 -8112.444} C_VEL
LIN {X 0,Y 460.602,Z 141.107,A -85,B 0,C 180,E1 -8115.997,E2 -8115.997} C_VEL
LIN {X 0,Y 460.569,Z 141.113,A -85,B 0,C 180,E1 -8119.615,E2 -8119.615} C_VEL
LIN {X 0,Y 460.511,Z 141.117,A -85,B 0,C 180,E1 -8122.428,E2 -8122.428} C_VEL
LIN {X 0,Y 460.547,Z 141.114,A -85,B 0,C 180,E1 -8125.796,E2 -8125.796} C_VEL
LIN {X 0,Y 460.55,Z 141.115,A -85,B 0,C 180,E1 -8128.233,E2 -8128.233} C_VEL
LIN {X 0,Y 460.52,Z 141.119,A -85,B 0,C 180,E1 -8131.282,E2 -8131.282} C_VEL
LIN {X 0,Y 460.522,Z 141.123,A -85,B 0,C 180,E1 -8134.503,E2 -8134.503} C_VEL
LIN {X 0,Y 460.5,Z 141.124,A -85,B 0,C 180,E1 -8137.623,E2 -8137.623} C_VEL
LIN {X 0,Y 460.54,Z 141.124,A -85,B 0,C 180,E1 -8140.269,E2 -8140.269} C_VEL
LIN {X 0,Y 460.498,Z 141.126,A -85,B 0,C 180,E1 -8143.375,E2 -8143.375} C_VEL
LIN {X 0,Y 460.498,Z 141.125,A -85,B 0,C 180,E1 -8146.624,E2 -8146.624} C_VEL
LIN {X 0,Y 460.587,Z 141.261,A -85,B 0,C 180,E1 -8148.729,E2 -8148.729} C_VEL
LIN {X 0,Y 461.864,Z 148.27,A -85,B 0,C 180,E1 -8150.275,E2 -8150.275} C_VEL
LIN {X 0,Y 461.862,Z 156.154,A -85,B 0,C 180,E1 -8151.919,E2 -8151.919} C_VEL
LIN {X 0,Y 461.682,Z 159.763,A -85,B 0,C 180,E1 -8152.662,E2 -8152.662} C_VEL
LIN {X 0,Y 464.885,Z 175.849,A -85,B 0,C 180,E1 -8153.076,E2 -8153.076} C_VEL
LIN {X 0,Y 463.955,Z 267.454,A -85,B 0,C 180,E1 -8154.541,E2 -8154.541} C_VEL
LIN {X 0,Y 463.684,Z 280.56,A -85,B 0,C 180,E1 -8154.931,E2 -8154.931} C_VEL
LIN {X 0,Y 463.306,Z 292.697,A -85,B 0,C 180,E1 -8155.462,E2 -8155.462} C_VEL
LIN {X 0,Y 462.873,Z 303.282,A -85,B 0,C 180,E1 -8156.077,E2 -8156.077} C_VEL
LIN {X 0,Y 462.394,Z 313.5,A -85,B 0,C 180,E1 -8156.827,E2 -8156.827} C_VEL
LIN {X 0,Y 461.81,Z 324.264,A -85,B 0,C 180,E1 -8157.816,E2 -8157.816} C_VEL
LIN {X 0,Y 461.313,Z 333.878,A -85,B 0,C 180,E1 -8158.91,E2 -8158.91} C_VEL
LIN {X 0,Y 460.411,Z 337.994,A -85,B 0,C 180,E1 -8159.428,E2 -8159.428} C_VEL
LIN {X 0,Y 457.203,Z 344.36,A -85,B 0,C 180,E1 -8160.293,E2 -8160.293} C_VEL
LIN {X 0,Y 454.041,Z 350.075,A -85,B 0,C 180,E1 -8161.232,E2 -8161.232} C_VEL
LIN {X 0,Y 453.222,Z 353.167,A -85,B 0,C 180,E1 -8161.86,E2 -8161.86} C_VEL
LIN {X 0,Y 452.937,Z 358.912,A -85,B 0,C 180,E1 -8163.258,E2 -8163.258} C_VEL
LIN {X 0,Y 452.707,Z 363.578,A -85,B 0,C 180,E1 -8164.728,E2 -8164.728} C_VEL
LIN {X 0,Y 452.574,Z 367.336,A -85,B 0,C 180,E1 -8166.376,E2 -8166.376} C_VEL
LIN {X 0,Y 452.466,Z 368.586,A -85,B 0,C 180,E1 -8167.15,E2 -8167.15} C_VEL
LIN {X 0,Y 452.398,Z 370.178,A -85,B 0,C 180,E1 -8168.763,E2 -8168.763} C_VEL
LIN {X 0,Y 452.377,Z 370.553,A -85,B 0,C 180,E1 -8170.014,E2 -8170.014} C_VEL
LIN {X 0,Y 452.406,Z 370.057,A -85,B 0,C 180,E1 -8171.371,E2 -8171.371} C_VEL
LIN {X 0,Y 452.454,Z 368.49,A -85,B 0,C 180,E1 -8172.835,E2 -8172.835} C_VEL
LIN {X 0,Y 452.611,Z 365.792,A -85,B 0,C 180,E1 -8174.303,E2 -8174.303} C_VEL
LIN {X 0,Y 452.744,Z 362.371,A -85,B 0,C 180,E1 -8175.619,E2 -8175.619} C_VEL
LIN {X 0,Y 452.929,Z 357.645,A -85,B 0,C 180,E1 -8176.998,E2 -8176.998} C_VEL
LIN {X 0,Y 453.199,Z 351.639,A -85,B 0,C 180,E1 -8178.37,E2 -8178.37} C_VEL
LIN {X 0,Y 453.594,Z 344.145,A -85,B 0,C 180,E1 -8179.736,E2 -8179.736} C_VEL
LIN {X 0,Y 453.994,Z 336.515,A -85,B 0,C 180,E1 -8180.87,E2 -8180.87} C_VEL
LIN {X 0,Y 454.501,Z 327.269,A -85,B 0,C 180,E1 -8182,E2 -8182} C_VEL
LIN {X 0,Y 455.064,Z 316.958,A -85,B 0,C 180,E1 -8183.014,E2 -8183.014} C_VEL
LIN {X 0,Y 455.62,Z 305.521,A -85,B 0,C 180,E1 -8183.913,E2 -8183.913} C_VEL
LIN {X 0,Y 456.094,Z 293.654,A -85,B 0,C 180,E1 -8184.64,E2 -8184.64} C_VEL
LIN {X 0,Y 456.413,Z 281.352,A -85,B 0,C 180,E1 -8185.197,E2 -8185.197} C_VEL
LIN {X 0,Y 456.724,Z 268.695,A -85,B 0,C 180,E1 -8185.587,E2 -8185.587} C_VEL
LIN {X 0,Y 456.978,Z 241.205,A -85,B 0,C 180,E1 -8186.059,E2 -8186.059} C_VEL
LIN {X 0,Y 457.464,Z 174.918,A -85,B 0,C 180,E1 -8187.114,E2 -8187.114} C_VEL
LIN {X 0,Y 454.488,Z 159.809,A -85,B 0,C 180,E1 -8187.48,E2 -8187.48} C_VEL
LIN {X 0,Y 454.735,Z 148.857,A -85,B 0,C 180,E1 -8189.779,E2 -8189.779} C_VEL
LIN {X 0,Y 453.623,Z 141.982,A -85,B 0,C 180,E1 -8191.332,E2 -8191.332} C_VEL
LIN {X 0,Y 453.697,Z 141.973,A -85,B 0,C 180,E1 -8192.664,E2 -8192.664} C_VEL
LIN {X 0,Y 453.629,Z 141.979,A -85,B 0,C 180,E1 -8196.226,E2 -8196.226} C_VEL
LIN {X 0,Y 453.553,Z 141.984,A -85,B 0,C 180,E1 -8198.914,E2 -8198.914} C_VEL
LIN {X 0,Y 453.56,Z 141.984,A -85,B 0,C 180,E1 -8202.529,E2 -8202.529} C_VEL
LIN {X 0,Y 453.481,Z 141.995,A -85,B 0,C 180,E1 -8206.199,E2 -8206.199} C_VEL
LIN {X 0,Y 453.481,Z 141.994,A -85,B 0,C 180,E1 -8209.028,E2 -8209.028} C_VEL
LIN {X 0,Y 453.462,Z 141.999,A -85,B 0,C 180,E1 -8211.837,E2 -8211.837} C_VEL
LIN {X 0,Y 453.445,Z 141.998,A -85,B 0,C 180,E1 -8214.739,E2 -8214.739} C_VEL
LIN {X 0,Y 453.452,Z 141.998,A -85,B 0,C 180,E1 -8217.942,E2 -8217.942} C_VEL
LIN {X 0,Y 453.443,Z 141.999,A -85,B 0,C 180,E1 -8220.762,E2 -8220.762} C_VEL
LIN {X 0,Y 453.451,Z 141.998,A -85,B 0,C 180,E1 -8223.915,E2 -8223.915} C_VEL
LIN {X 0,Y 453.431,Z 142.007,A -85,B 0,C 180,E1 -8227.192,E2 -8227.192} C_VEL
LIN {X 0,Y 453.465,Z 141.997,A -85,B 0,C 180,E1 -8230.613,E2 -8230.613} C_VEL
LIN {X 0,Y 453.479,Z 141.996,A -85,B 0,C 180,E1 -8234.529,E2 -8234.529} C_VEL
LIN {X 0,Y 453.434,Z 141.999,A -85,B 0,C 180,E1 -8238.072,E2 -8238.072} C_VEL
LIN {X 0,Y 453.438,Z 142.006,A -85,B 0,C 180,E1 -8240.803,E2 -8240.803} C_VEL
LIN {X 0,Y 453.442,Z 141.998,A -85,B 0,C 180,E1 -8243.917,E2 -8243.917} C_VEL
LIN {X 0,Y 453.465,Z 142.001,A -85,B 0,C 180,E1 -8246.817,E2 -8246.817} C_VEL
LIN {X 0,Y 453.448,Z 142.001,A -85,B 0,C 180,E1 -8250.267,E2 -8250.267} C_VEL
LIN {X 0,Y 453.424,Z 142,A -85,B 0,C 180,E1 -8253.289,E2 -8253.289} C_VEL
LIN {X 0,Y 453.473,Z 141.999,A -85,B 0,C 180,E1 -8256.238,E2 -8256.238} C_VEL
LIN {X 0,Y 453.439,Z 141.999,A -85,B 0,C 180,E1 -8259.116,E2 -8259.116} C_VEL
LIN {X 0,Y 453.459,Z 141.999,A -85,B 0,C 180,E1 -8261.943,E2 -8261.943} C_VEL
LIN {X 0,Y 453.489,Z 141.994,A -85,B 0,C 180,E1 -8264.725,E2 -8264.725} C_VEL
LIN {X 0,Y 453.568,Z 141.983,A -85,B 0,C 180,E1 -8267.472,E2 -8267.472} C_VEL
LIN {X 0,Y 453.559,Z 141.983,A -85,B 0,C 180,E1 -8271.086,E2 -8271.086} C_VEL
LIN {X 0,Y 453.639,Z 141.978,A -85,B 0,C 180,E1 -8273.775,E2 -8273.775} C_VEL
LIN {X 0,Y 453.705,Z 141.967,A -85,B 0,C 180,E1 -8277.337,E2 -8277.337} C_VEL
LIN {X 0,Y 453.772,Z 141.963,A -85,B 0,C 180,E1 -8280,E2 -8280} C_VEL
LIN {X 0,Y 453.706,Z 141.965,A -85,B 0,C 180,E1 -8282.664,E2 -8282.664} C_VEL
LIN {X 0,Y 453.633,Z 141.976,A -85,B 0,C 180,E1 -8286.226,E2 -8286.226} C_VEL
LIN {X 0,Y 453.566,Z 141.983,A -85,B 0,C 180,E1 -8288.914,E2 -8288.914} C_VEL
LIN {X 0,Y 453.57,Z 141.982,A -85,B 0,C 180,E1 -8292.529,E2 -8292.529} C_VEL
LIN {X 0,Y 453.506,Z 141.99,A -85,B 0,C 180,E1 -8296.198,E2 -8296.198} C_VEL
LIN {X 0,Y 453.522,Z 141.992,A -85,B 0,C 180,E1 -8299.039,E2 -8299.039} C_VEL
LIN {X 0,Y 453.478,Z 141.995,A -85,B 0,C 180,E1 -8301.837,E2 -8301.837} C_VEL
LIN {X 0,Y 453.472,Z 141.996,A -85,B 0,C 180,E1 -8304.737,E2 -8304.737} C_VEL
LIN {X 0,Y 453.466,Z 141.995,A -85,B 0,C 180,E1 -8307.942,E2 -8307.942} C_VEL
LIN {X 0,Y 453.458,Z 142,A -85,B 0,C 180,E1 -8310.761,E2 -8310.761} C_VEL
LIN {X 0,Y 453.471,Z 141.994,A -85,B 0,C 180,E1 -8313.914,E2 -8313.914} C_VEL
LIN {X 0,Y 453.454,Z 142.001,A -85,B 0,C 180,E1 -8317.19,E2 -8317.19} C_VEL
LIN {X 0,Y 453.474,Z 141.999,A -85,B 0,C 180,E1 -8320.612,E2 -8320.612} C_VEL
LIN {X 0,Y 453.485,Z 141.998,A -85,B 0,C 180,E1 -8324.528,E2 -8324.528} C_VEL
LIN {X 0,Y 453.44,Z 142,A -85,B 0,C 180,E1 -8328.071,E2 -8328.071} C_VEL
LIN {X 0,Y 453.452,Z 142.001,A -85,B 0,C 180,E1 -8330.801,E2 -8330.801} C_VEL
LIN {X 0,Y 453.455,Z 141.998,A -85,B 0,C 180,E1 -8333.917,E2 -8333.917} C_VEL
LIN {X 0,Y 453.478,Z 141.994,A -85,B 0,C 180,E1 -8337.15,E2 -8337.15} C_VEL
LIN {X 0,Y 453.466,Z 142.003,A -85,B 0,C 180,E1 -8340.267,E2 -8340.267} C_VEL
LIN {X 0,Y 453.498,Z 142.037,A -85,B 0,C 180,E1 -8343.678,E2 -8343.678} C_VEL
LIN {X 0,Y 455.754,Z 153.694,A -85,B 0,C 180,E1 -8345.935,E2 -8345.935} C_VEL
LIN {X 0,Y 455.497,Z 163.21,A -85,B 0,C 180,E1 -8347.654,E2 -8347.654} C_VEL
LIN {X 0,Y 454.564,Z 183.689,A -85,B 0,C 180,E1 -8351.287,E2 -8351.287} C_VEL
LIN {X 0,Y 454.285,Z 190.812,A -85,B 0,C 180,E1 -8352.54,E2 -8352.54} C_VEL
LIN {X 0,Y 457.391,Z 212.181,A -85,B 0,C 180,E1 -8353.001,E2 -8353.001} C_VEL
LIN {X 0,Y 456.597,Z 299.29,A -85,B 0,C 180,E1 -8354.402,E2 -8354.402} C_VEL
LIN {X 0,Y 456.236,Z 312.537,A -85,B 0,C 180,E1 -8354.79,E2 -8354.79} C_VEL
LIN {X 0,Y 455.758,Z 324.705,A -85,B 0,C 180,E1 -8355.317,E2 -8355.317} C_VEL
LIN {X 0,Y 455.192,Z 336.992,A -85,B 0,C 180,E1 -8356.04,E2 -8356.04} C_VEL
LIN {X 0,Y 454.612,Z 349.064,A -85,B 0,C 180,E1 -8356.972,E2 -8356.972} C_VEL
LIN {X 0,Y 454.13,Z 359.086,A -85,B 0,C 180,E1 -8357.941,E2 -8357.941} C_VEL
LIN {X 0,Y 453.625,Z 368.495,A -85,B 0,C 180,E1 -8359.059,E2 -8359.059} C_VEL
LIN {X 0,Y 453.166,Z 377.588,A -85,B 0,C 180,E1 -8360.403,E2 -8360.403} C_VEL
LIN {X 0,Y 452.851,Z 384.914,A -85,B 0,C 180,E1 -8361.746,E2 -8361.746} C_VEL
LIN {X 0,Y 452.675,Z 389.867,A -85,B 0,C 180,E1 -8362.865,E2 -8362.865} C_VEL
LIN {X 0,Y 452.532,Z 394.675,A -85,B 0,C 180,E1 -8364.206,E2 -8364.206} C_VEL
LIN {X 0,Y 452.485,Z 398.356,A -85,B 0,C 180,E1 -8365.546,E2 -8365.546} C_VEL
LIN {X 0,Y 452.483,Z 400.257,A -85,B 0,C 180,E1 -8366.438,E2 -8366.438} C_VEL
LIN {X 0,Y 452.508,Z 401.699,A -85,B 0,C 180,E1 -8367.329,E2 -8367.329} C_VEL
LIN {X 0,Y 452.46,Z 403.343,A -85,B 0,C 180,E1 -8369.11,E2 -8369.11} C_VEL
LIN {X 0,Y 452.47,Z 403.583,A -85,B 0,C 180,E1 -8370,E2 -8370} C_VEL
LIN {X 0,Y 452.433,Z 403.395,A -85,B 0,C 180,E1 -8370.89,E2 -8370.89} C_VEL
LIN {X 0,Y 452.508,Z 401.816,A -85,B 0,C 180,E1 -8372.67,E2 -8372.67} C_VEL
LIN {X 0,Y 452.481,Z 400.434,A -85,B 0,C 180,E1 -8373.562,E2 -8373.562} C_VEL
LIN {X 0,Y 452.542,Z 397.518,A -85,B 0,C 180,E1 -8374.9,E2 -8374.9} C_VEL
LIN {X 0,Y 452.555,Z 393.275,A -85,B 0,C 180,E1 -8376.331,E2 -8376.331} C_VEL
LIN {X 0,Y 452.776,Z 388.491,A -85,B 0,C 180,E1 -8377.581,E2 -8377.581} C_VEL
LIN {X 0,Y 453.031,Z 382.115,A -85,B 0,C 180,E1 -8378.924,E2 -8378.924} C_VEL
LIN {X 0,Y 453.386,Z 374.143,A -85,B 0,C 180,E1 -8380.269,E2 -8380.269} C_VEL
LIN {X 0,Y 454.003,Z 364.247,A -85,B 0,C 180,E1 -8381.609,E2 -8381.609} C_VEL
LIN {X 0,Y 454.486,Z 354.799,A -85,B 0,C 180,E1 -8382.644,E2 -8382.644} C_VEL
LIN {X 0,Y 455.073,Z 343.686,A -85,B 0,C 180,E1 -8383.622,E2 -8383.622} C_VEL
LIN {X 0,Y 455.676,Z 332.536,A -85,B 0,C 180,E1 -8384.401,E2 -8384.401} C_VEL
LIN {X 0,Y 456.313,Z 320.141,A -85,B 0,C 180,E1 -8385.064,E2 -8385.064} C_VEL
LIN {X 0,Y 456.776,Z 306.972,A -85,B 0,C 180,E1 -8385.563,E2 -8385.563} C_VEL
LIN {X 0,Y 457.17,Z 294.274,A -85,B 0,C 180,E1 -8385.864,E2 -8385.864} C_VEL
LIN {X 0,Y 457.733,Z 211.247,A -85,B 0,C 180,E1 -8387.205,E2 -8387.205} C_VEL
LIN {X 0,Y 454.442,Z 190.39,A -85,B 0,C 180,E1 -8387.703,E2 -8387.703} C_VEL
LIN {X 0,Y 455.114,Z 174.321,A -85,B 0,C 180,E1 -8390.568,E2 -8390.568} C_VEL
LIN {X 0,Y 456.065,Z 157.392,A -85,B 0,C 180,E1 -8393.62,E2 -8393.62} C_VEL
LIN {X 0,Y 455.687,Z 152.75,A -85,B 0,C 180,E1 -8394.501,E2 -8394.501} C_VEL
LIN {X 0,Y 453.475,Z 142,A -85,B 0,C 180,E1 -8396.708,E2 -8396.708} C_VEL
LIN {X 0,Y 453.471,Z 142.002,A -85,B 0,C 180,E1 -8399.784,E2 -8399.784} C_VEL
LIN {X 0,Y 453.483,Z 141.999,A -85,B 0,C 180,E1 -8403.187,E2 -8403.187} C_VEL
LIN {X 0,Y 453.45,Z 141.999,A -85,B 0,C 180,E1 -8406.298,E2 -8406.298} C_VEL
LIN {X 0,Y 453.445,Z 142.003,A -85,B 0,C 180,E1 -8409.455,E2 -8409.455} C_VEL
LIN {X 0,Y 453.438,Z 142.001,A -85,B 0,C 180,E1 -8411.929,E2 -8411.929} C_VEL
LIN {X 0,Y 453.483,Z 141.997,A -85,B 0,C 180,E1 -8415.471,E2 -8415.471} C_VEL
LIN {X 0,Y 453.469,Z 141.998,A -85,B 0,C 180,E1 -8419.388,E2 -8419.388} C_VEL
LIN {X 0,Y 453.434,Z 142.003,A -85,B 0,C 180,E1 -8422.808,E2 -8422.808} C_VEL
LIN {X 0,Y 453.454,Z 141.995,A -85,B 0,C 180,E1 -8426.085,E2 -8426.085} C_VEL
LIN {X 0,Y 453.449,Z 141.996,A -85,B 0,C 180,E1 -8429.238,E2 -8429.238} C_VEL
LIN {X 0,Y 453.471,Z 141.999,A -85,B 0,C 180,E1 -8432.293,E2 -8432.293} C_VEL
LIN {X 0,Y 453.463,Z 141.996,A -85,B 0,C 180,E1 -8435.262,E2 -8435.262} C_VEL
LIN {X 0,Y 453.476,Z 141.997,A -85,B 0,C 180,E1 -8438.417,E2 -8438.417} C_VEL
LIN {X 0,Y 453.459,Z 141.997,A -85,B 0,C 180,E1 -8441.942,E2 -8441.942} C_VEL
LIN {X 0,Y 453.52,Z 141.99,A -85,B 0,C 180,E1 -8444.725,E2 -8444.725} C_VEL
LIN {X 0,Y 453.548,Z 141.989,A -85,B 0,C 180,E1 -8448.378,E2 -8448.378} C_VEL
LIN {X 0,Y 453.573,Z 141.98,A -85,B 0,C 180,E1 -8451.086,E2 -8451.086} C_VEL
LIN {X 0,Y 453.64,Z 141.978,A -85,B 0,C 180,E1 -8453.774,E2 -8453.774} C_VEL
LIN {X 0,Y 453.707,Z 141.961,A -85,B 0,C 180,E1 -8457.336,E2 -8457.336} C_VEL
LIN {X 0,Y 453.794,Z 141.955,A -85,B 0,C 180,E1 -8460,E2 -8460} C_VEL
LIN {X 0,Y 453.736,Z 141.96,A -85,B 0,C 180,E1 -8462.663,E2 -8462.663} C_VEL
LIN {X 0,Y 453.646,Z 141.97,A -85,B 0,C 180,E1 -8466.225,E2 -8466.225} C_VEL
LIN {X 0,Y 453.586,Z 141.984,A -85,B 0,C 180,E1 -8468.913,E2 -8468.913} C_VEL
LIN {X 0,Y 453.566,Z 141.984,A -85,B 0,C 180,E1 -8472.528,E2 -8472.528} C_VEL
LIN {X 0,Y 453.546,Z 141.986,A -85,B 0,C 180,E1 -8476.195,E2 -8476.195} C_VEL
LIN {X 0,Y 453.518,Z 141.993,A -85,B 0,C 180,E1 -8479.039,E2 -8479.039} C_VEL
LIN {X 0,Y 453.477,Z 141.991,A -85,B 0,C 180,E1 -8481.836,E2 -8481.836} C_VEL
LIN {X 0,Y 453.496,Z 141.997,A -85,B 0,C 180,E1 -8484.735,E2 -8484.735} C_VEL
LIN {X 0,Y 453.529,Z 141.988,A -85,B 0,C 180,E1 -8487.958,E2 -8487.958} C_VEL
LIN {X 0,Y 453.465,Z 141.997,A -85,B 0,C 180,E1 -8491.524,E2 -8491.524} C_VEL
LIN {X 0,Y 453.481,Z 141.999,A -85,B 0,C 180,E1 -8494.776,E2 -8494.776} C_VEL
LIN {X 0,Y 453.463,Z 142.003,A -85,B 0,C 180,E1 -8498.311,E2 -8498.311} C_VEL
LIN {X 0,Y 453.493,Z 142.002,A -85,B 0,C 180,E1 -8500.608,E2 -8500.608} C_VEL
LIN {X 0,Y 453.454,Z 142.004,A -85,B 0,C 180,E1 -8503.244,E2 -8503.244} C_VEL
LIN {X 0,Y 453.464,Z 142.001,A -85,B 0,C 180,E1 -8505.779,E2 -8505.779} C_VEL
LIN {X 0,Y 453.55,Z 142.116,A -85,B 0,C 180,E1 -8508.491,E2 -8508.491} C_VEL
LIN {X 0,Y 455.022,Z 150.571,A -85,B 0,C 180,E1 -8510.378,E2 -8510.378} C_VEL
LIN {X 0,Y 454.762,Z 160.087,A -85,B 0,C 180,E1 -8512.372,E2 -8512.372} C_VEL
LIN {X 0,Y 458.177,Z 176.766,A -85,B 0,C 180,E1 -8512.801,E2 -8512.801} C_VEL
LIN {X 0,Y 457.178,Z 266.737,A -85,B 0,C 180,E1 -8514.256,E2 -8514.256} C_VEL
LIN {X 0,Y 456.922,Z 279.73,A -85,B 0,C 180,E1 -8514.637,E2 -8514.637} C_VEL
LIN {X 0,Y 456.517,Z 292.022,A -85,B 0,C 180,E1 -8515.171,E2 -8515.171} C_VEL
LIN {X 0,Y 456.069,Z 302.457,A -85,B 0,C 180,E1 -8515.774,E2 -8515.774} C_VEL
LIN {X 0,Y 455.551,Z 312.804,A -85,B 0,C 180,E1 -8516.528,E2 -8516.528} C_VEL
LIN {X 0,Y 454.936,Z 323.787,A -85,B 0,C 180,E1 -8517.532,E2 -8517.532} C_VEL
LIN {X 0,Y 454.44,Z 332.684,A -85,B 0,C 180,E1 -8518.537,E2 -8518.537} C_VEL
LIN {X 0,Y 453.901,Z 341.577,A -85,B 0,C 180,E1 -8519.763,E2 -8519.763} C_VEL
LIN {X 0,Y 453.499,Z 349.073,A -85,B 0,C 180,E1 -8521.034,E2 -8521.034} C_VEL
LIN {X 0,Y 453.222,Z 353.167,A -85,B 0,C 180,E1 -8521.86,E2 -8521.86} C_VEL
LIN {X 0,Y 452.422,Z 356.081,A -85,B 0,C 180,E1 -8522.507,E2 -8522.507} C_VEL
LIN {X 0,Y 449.349,Z 360.387,A -85,B 0,C 180,E1 -8523.575,E2 -8523.575} C_VEL
LIN {X 0,Y 446.303,Z 363.995,A -85,B 0,C 180,E1 -8524.693,E2 -8524.693} C_VEL
LIN {X 0,Y 445.556,Z 365.769,A -85,B 0,C 180,E1 -8525.411,E2 -8525.411} C_VEL
LIN {X 0,Y 445.441,Z 368.355,A -85,B 0,C 180,E1 -8526.769,E2 -8526.769} C_VEL
LIN {X 0,Y 445.339,Z 369.651,A -85,B 0,C 180,E1 -8527.744,E2 -8527.744} C_VEL
LIN {X 0,Y 445.315,Z 370.434,A -85,B 0,C 180,E1 -8528.716,E2 -8528.716} C_VEL
LIN {X 0,Y 445.275,Z 370.775,A -85,B 0,C 180,E1 -8529.682,E2 -8529.682} C_VEL
LIN {X 0,Y 445.306,Z 370.384,A -85,B 0,C 180,E1 -8531.251,E2 -8531.251} C_VEL
LIN {X 0,Y 445.334,Z 369.14,A -85,B 0,C 180,E1 -8532.552,E2 -8532.552} C_VEL
LIN {X 0,Y 445.514,Z 366.357,A -85,B 0,C 180,E1 -8534.21,E2 -8534.21} C_VEL
LIN {X 0,Y 445.699,Z 362.118,A -85,B 0,C 180,E1 -8535.853,E2 -8535.853} C_VEL
LIN {X 0,Y 445.912,Z 357.251,A -85,B 0,C 180,E1 -8537.253,E2 -8537.253} C_VEL
LIN {X 0,Y 446.204,Z 351.097,A -85,B 0,C 180,E1 -8538.645,E2 -8538.645} C_VEL
LIN {X 0,Y 446.622,Z 343.44,A -85,B 0,C 180,E1 -8540.032,E2 -8540.032} C_VEL
LIN {X 0,Y 447.061,Z 335.606,A -85,B 0,C 180,E1 -8541.184,E2 -8541.184} C_VEL
LIN {X 0,Y 447.616,Z 326.012,A -85,B 0,C 180,E1 -8542.331,E2 -8542.331} C_VEL
LIN {X 0,Y 448.247,Z 315.335,A -85,B 0,C 180,E1 -8543.36,E2 -8543.36} C_VEL
LIN {X 0,Y 448.798,Z 303.429,A -85,B 0,C 180,E1 -8544.271,E2 -8544.271} C_VEL
LIN {X 0,Y 449.253,Z 290.699,A -85,B 0,C 180,E1 -8545.008,E2 -8545.008} C_VEL
LIN {X 0,Y 449.632,Z 277.912,A -85,B 0,C 180,E1 -8545.546,E2 -8545.546} C_VEL
LIN {X 0,Y 449.887,Z 265.499,A -85,B 0,C 180,E1 -8545.885,E2 -8545.885} C_VEL
LIN {X 0,Y 450.649,Z 175.928,A -85,B 0,C 180,E1 -8547.343,E2 -8547.343} C_VEL
LIN {X 0,Y 447.532,Z 160.022,A -85,B 0,C 180,E1 -8547.736,E2 -8547.736} C_VEL
LIN {X 0,Y 447.778,Z 150.42,A -85,B 0,C 180,E1 -8549.775,E2 -8549.775} C_VEL
LIN {X 0,Y 446.611,Z 142.856,A -85,B 0,C 180,E1 -8551.465,E2 -8551.465} C_VEL
LIN {X 0,Y 446.646,Z 142.851,A -85,B 0,C 180,E1 -8552.706,E2 -8552.706} C_VEL
LIN {X 0,Y 446.599,Z 142.853,A -85,B 0,C 180,E1 -8556.325,E2 -8556.325} C_VEL
LIN {X 0,Y 446.504,Z 142.863,A -85,B 0,C 180,E1 -8559.056,E2 -8559.056} C_VEL
LIN {X 0,Y 446.488,Z 142.864,A -85,B 0,C 180,E1 -8562.731,E2 -8562.731} C_VEL
LIN {X 0,Y 446.45,Z 142.871,A -85,B 0,C 180,E1 -8566.209,E2 -8566.209} C_VEL
LIN {X 0,Y 446.423,Z 142.876,A -85,B 0,C 180,E1 -8569.306,E2 -8569.306} C_VEL
LIN {X 0,Y 446.399,Z 142.876,A -85,B 0,C 180,E1 -8572.201,E2 -8572.201} C_VEL
LIN {X 0,Y 446.401,Z 142.879,A -85,B 0,C 180,E1 -8575.156,E2 -8575.156} C_VEL
LIN {X 0,Y 446.411,Z 142.874,A -85,B 0,C 180,E1 -8578.184,E2 -8578.184} C_VEL
LIN {X 0,Y 446.385,Z 142.885,A -85,B 0,C 180,E1 -8581.303,E2 -8581.303} C_VEL
LIN {X 0,Y 446.409,Z 142.875,A -85,B 0,C 180,E1 -8584.525,E2 -8584.525} C_VEL
LIN {X 0,Y 446.392,Z 142.876,A -85,B 0,C 180,E1 -8588.076,E2 -8588.076} C_VEL
LIN {X 0,Y 446.395,Z 142.879,A -85,B 0,C 180,E1 -8591.395,E2 -8591.395} C_VEL
LIN {X 0,Y 446.448,Z 142.875,A -85,B 0,C 180,E1 -8595.105,E2 -8595.105} C_VEL
LIN {X 0,Y 446.399,Z 142.88,A -85,B 0,C 180,E1 -8598.606,E2 -8598.606} C_VEL
LIN {X 0,Y 446.397,Z 142.876,A -85,B 0,C 180,E1 -8601.925,E2 -8601.925} C_VEL
LIN {X 0,Y 446.413,Z 142.874,A -85,B 0,C 180,E1 -8605.476,E2 -8605.476} C_VEL
LIN {X 0,Y 446.389,Z 142.883,A -85,B 0,C 180,E1 -8608.698,E2 -8608.698} C_VEL
LIN {X 0,Y 446.401,Z 142.876,A -85,B 0,C 180,E1 -8611.843,E2 -8611.843} C_VEL
LIN {X 0,Y 446.408,Z 142.877,A -85,B 0,C 180,E1 -8614.845,E2 -8614.845} C_VEL
LIN {X 0,Y 446.444,Z 142.876,A -85,B 0,C 180,E1 -8618.248,E2 -8618.248} C_VEL
LIN {X 0,Y 446.412,Z 142.875,A -85,B 0,C 180,E1 -8621.648,E2 -8621.648} C_VEL
LIN {X 0,Y 446.431,Z 142.876,A -85,B 0,C 180,E1 -8624.478,E2 -8624.478} C_VEL
LIN {X 0,Y 446.52,Z 142.861,A -85,B 0,C 180,E1 -8627.385,E2 -8627.385} C_VEL
LIN {X 0,Y 446.51,Z 142.862,A -85,B 0,C 180,E1 -8630.945,E2 -8630.945} C_VEL
LIN {X 0,Y 446.609,Z 142.853,A -85,B 0,C 180,E1 -8633.676,E2 -8633.676} C_VEL
LIN {X 0,Y 446.655,Z 142.845,A -85,B 0,C 180,E1 -8637.295,E2 -8637.295} C_VEL
LIN {X 0,Y 446.722,Z 142.841,A -85,B 0,C 180,E1 -8640,E2 -8640} C_VEL
LIN {X 0,Y 446.655,Z 142.843,A -85,B 0,C 180,E1 -8642.706,E2 -8642.706} C_VEL
LIN {X 0,Y 446.604,Z 142.851,A -85,B 0,C 180,E1 -8646.325,E2 -8646.325} C_VEL
LIN {X 0,Y 446.517,Z 142.862,A -85,B 0,C 180,E1 -8649.056,E2 -8649.056} C_VEL
LIN {X 0,Y 446.527,Z 142.86,A -85,B 0,C 180,E1 -8652.73,E2 -8652.73} C_VEL
LIN {X 0,Y 446.459,Z 142.868,A -85,B 0,C 180,E1 -8656.209,E2 -8656.209} C_VEL
LIN {X 0,Y 446.472,Z 142.873,A -85,B 0,C 180,E1 -8659.304,E2 -8659.304} C_VEL
LIN {X 0,Y 446.418,Z 142.873,A -85,B 0,C 180,E1 -8662.2,E2 -8662.2} C_VEL
LIN {X 0,Y 446.424,Z 142.879,A -85,B 0,C 180,E1 -8665.155,E2 -8665.155} C_VEL
LIN {X 0,Y 446.421,Z 142.873,A -85,B 0,C 180,E1 -8668.183,E2 -8668.183} C_VEL
LIN {X 0,Y 446.397,Z 142.88,A -85,B 0,C 180,E1 -8671.302,E2 -8671.302} C_VEL
LIN {X 0,Y 446.426,Z 142.874,A -85,B 0,C 180,E1 -8674.524,E2 -8674.524} C_VEL
LIN {X 0,Y 446.415,Z 142.874,A -85,B 0,C 180,E1 -8678.078,E2 -8678.078} C_VEL
LIN {X 0,Y 446.404,Z 142.876,A -85,B 0,C 180,E1 -8681.394,E2 -8681.394} C_VEL
LIN {X 0,Y 446.453,Z 142.871,A -85,B 0,C 180,E1 -8685.104,E2 -8685.104} C_VEL
LIN {X 0,Y 446.404,Z 142.882,A -85,B 0,C 180,E1 -8688.606,E2 -8688.606} C_VEL
LIN {X 0,Y 446.414,Z 142.875,A -85,B 0,C 180,E1 -8691.922,E2 -8691.922} C_VEL
LIN {X 0,Y 446.425,Z 142.872,A -85,B 0,C 180,E1 -8695.476,E2 -8695.476} C_VEL
LIN {X 0,Y 446.418,Z 142.879,A -85,B 0,C 180,E1 -8698.699,E2 -8698.699} C_VEL
LIN {X 0,Y 446.427,Z 142.878,A -85,B 0,C 180,E1 -8701.836,E2 -8701.836} C_VEL
LIN {X 0,Y 446.441,Z 142.893,A -85,B 0,C 180,E1 -8703.481,E2 -8703.481} C_VEL
LIN {X 0,Y 448.881,Z 155.634,A -85,B 0,C 180,E1 -8705.978,E2 -8705.978} C_VEL
LIN {X 0,Y 448.205,Z 170.136,A -85,B 0,C 180,E1 -8708.619,E2 -8708.619} C_VEL
LIN {X 0,Y 447.363,Z 188.668,A -85,B 0,C 180,E1 -8711.948,E2 -8711.948} C_VEL
LIN {X 0,Y 447.336,Z 190.876,A -85,B 0,C 180,E1 -8712.3,E2 -8712.3} C_VEL
LIN {X 0,Y 450.531,Z 213.717,A -85,B 0,C 180,E1 -8712.789,E2 -8712.789} C_VEL
LIN {X 0,Y 449.721,Z 299.322,A -85,B 0,C 180,E1 -8714.186,E2 -8714.186} C_VEL
LIN {X 0,Y 449.328,Z 313.256,A -85,B 0,C 180,E1 -8714.608,E2 -8714.608} C_VEL
LIN {X 0,Y 448.832,Z 325.189,A -85,B 0,C 180,E1 -8715.143,E2 -8715.143} C_VEL
LIN {X 0,Y 448.277,Z 336.465,A -85,B 0,C 180,E1 -8715.82,E2 -8715.82} C_VEL
LIN {X 0,Y 447.681,Z 347.857,A -85,B 0,C 180,E1 -8716.702,E2 -8716.702} C_VEL
LIN {X 0,Y 447.087,Z 358.643,A -85,B 0,C 180,E1 -8717.748,E2 -8717.748} C_VEL
LIN {X 0,Y 446.639,Z 368.101,A -85,B 0,C 180,E1 -8718.886,E2 -8718.886} C_VEL
LIN {X 0,Y 446.133,Z 377.217,A -85,B 0,C 180,E1 -8720.25,E2 -8720.25} C_VEL
LIN {X 0,Y 445.796,Z 384.563,A -85,B 0,C 180,E1 -8721.615,E2 -8721.615} C_VEL
LIN {X 0,Y 445.603,Z 389.534,A -85,B 0,C 180,E1 -8722.751,E2 -8722.751} C_VEL
LIN {X 0,Y 445.445,Z 393.954,A -85,B 0,C 180,E1 -8723.986,E2 -8723.986} C_VEL
LIN {X 0,Y 445.411,Z 398.055,A -85,B 0,C 180,E1 -8725.475,E2 -8725.475} C_VEL
LIN {X 0,Y 445.383,Z 399.962,A -85,B 0,C 180,E1 -8726.381,E2 -8726.381} C_VEL
LIN {X 0,Y 445.433,Z 401.418,A -85,B 0,C 180,E1 -8727.287,E2 -8727.287} C_VEL
LIN {X 0,Y 445.369,Z 403.074,A -85,B 0,C 180,E1 -8729.096,E2 -8729.096} C_VEL
LIN {X 0,Y 445.375,Z 403.32,A -85,B 0,C 180,E1 -8730,E2 -8730} C_VEL
LIN {X 0,Y 445.344,Z 403.144,A -85,B 0,C 180,E1 -8730.904,E2 -8730.904} C_VEL
LIN {X 0,Y 445.433,Z 401.577,A -85,B 0,C 180,E1 -8732.713,E2 -8732.713} C_VEL
LIN {X 0,Y 445.38,Z 400.199,A -85,B 0,C 180,E1 -8733.619,E2 -8733.619} C_VEL
LIN {X 0,Y 445.47,Z 397.296,A -85,B 0,C 180,E1 -8734.978,E2 -8734.978} C_VEL
LIN {X 0,Y 445.456,Z 393.357,A -85,B 0,C 180,E1 -8736.341,E2 -8736.341} C_VEL
LIN {X 0,Y 445.708,Z 388.292,A -85,B 0,C 180,E1 -8737.702,E2 -8737.702} C_VEL
LIN {X 0,Y 445.976,Z 381.935,A -85,B 0,C 180,E1 -8739.067,E2 -8739.067} C_VEL
LIN {X 0,Y 446.349,Z 373.992,A -85,B 0,C 180,E1 -8740.432,E2 -8740.432} C_VEL
LIN {X 0,Y 446.926,Z 365.926,A -85,B 0,C 180,E1 -8741.566,E2 -8741.566} C_VEL
LIN {X 0,Y 447.455,Z 356.104,A -85,B 0,C 180,E1 -8742.703,E2 -8742.703} C_VEL
LIN {X 0,Y 448.086,Z 345.159,A -85,B 0,C 180,E1 -8743.723,E2 -8743.723} C_VEL
LIN {X 0,Y 448.821,Z 332.689,A -85,B 0,C 180,E1 -8744.625,E2 -8744.625} C_VEL
LIN {X 0,Y 449.48,Z 320.455,A -85,B 0,C 180,E1 -8745.299,E2 -8745.299} C_VEL
LIN {X 0,Y 449.939,Z 307.591,A -85,B 0,C 180,E1 -8745.805,E2 -8745.805} C_VEL
LIN {X 0,Y 450.424,Z 293.97,A -85,B 0,C 180,E1 -8746.137,E2 -8746.137} C_VEL
LIN {X 0,Y 451.001,Z 212.182,A -85,B 0,C 180,E1 -8747.48,E2 -8747.48} C_VEL
LIN {X 0,Y 447.49,Z 190.137,A -85,B 0,C 180,E1 -8748.014,E2 -8748.014} C_VEL
LIN {X 0,Y 448.428,Z 171.613,A -85,B 0,C 180,E1 -8751.37,E2 -8751.37} C_VEL
LIN {X 0,Y 449.191,Z 157.325,A -85,B 0,C 180,E1 -8754.004,E2 -8754.004} C_VEL
LIN {X 0,Y 447.33,Z 146.939,A -85,B 0,C 180,E1 -8756.098,E2 -8756.098} C_VEL
LIN {X 0,Y 446.443,Z 142.876,A -85,B 0,C 180,E1 -8756.987,E2 -8756.987} C_VEL
LIN {X 0,Y 446.428,Z 142.879,A -85,B 0,C 180,E1 -8760.25,E2 -8760.25} C_VEL
LIN {X 0,Y 446.426,Z 142.879,A -85,B 0,C 180,E1 -8763.449,E2 -8763.449} C_VEL
LIN {X 0,Y 446.4,Z 142.878,A -85,B 0,C 180,E1 -8766.746,E2 -8766.746} C_VEL
LIN {X 0,Y 446.4,Z 142.875,A -85,B 0,C 180,E1 -8770.203,E2 -8770.203} C_VEL
LIN {X 0,Y 446.387,Z 142.879,A -85,B 0,C 180,E1 -8773.594,E2 -8773.594} C_VEL
LIN {X 0,Y 446.389,Z 142.878,A -85,B 0,C 180,E1 -8776.152,E2 -8776.152} C_VEL
LIN {X 0,Y 446.399,Z 142.879,A -85,B 0,C 180,E1 -8779.087,E2 -8779.087} C_VEL
LIN {X 0,Y 446.389,Z 142.876,A -85,B 0,C 180,E1 -8782.119,E2 -8782.119} C_VEL
LIN {X 0,Y 446.412,Z 142.872,A -85,B 0,C 180,E1 -8785.475,E2 -8785.475} C_VEL
LIN {X 0,Y 446.39,Z 142.878,A -85,B 0,C 180,E1 -8788.697,E2 -8788.697} C_VEL
LIN {X 0,Y 446.403,Z 142.876,A -85,B 0,C 180,E1 -8791.842,E2 -8791.842} C_VEL
LIN {X 0,Y 446.414,Z 142.877,A -85,B 0,C 180,E1 -8794.845,E2 -8794.845} C_VEL
LIN {X 0,Y 446.445,Z 142.87,A -85,B 0,C 180,E1 -8798.247,E2 -8798.247} C_VEL
LIN {X 0,Y 446.412,Z 142.873,A -85,B 0,C 180,E1 -8801.647,E2 -8801.647} C_VEL
LIN {X 0,Y 446.46,Z 142.872,A -85,B 0,C 180,E1 -8804.478,E2 -8804.478} C_VEL
LIN {X 0,Y 446.519,Z 142.855,A -85,B 0,C 180,E1 -8807.384,E2 -8807.384} C_VEL
LIN {X 0,Y 446.521,Z 142.858,A -85,B 0,C 180,E1 -8810.944,E2 -8810.944} C_VEL
LIN {X 0,Y 446.61,Z 142.852,A -85,B 0,C 180,E1 -8813.675,E2 -8813.675} C_VEL
LIN {X 0,Y 446.656,Z 142.839,A -85,B 0,C 180,E1 -8817.294,E2 -8817.294} C_VEL
LIN {X 0,Y 446.764,Z 142.83,A -85,B 0,C 180,E1 -8820,E2 -8820} C_VEL
LIN {X 0,Y 446.683,Z 142.839,A -85,B 0,C 180,E1 -8822.705,E2 -8822.705} C_VEL
LIN {X 0,Y 446.615,Z 142.845,A -85,B 0,C 180,E1 -8826.324,E2 -8826.324} C_VEL
LIN {X 0,Y 446.533,Z 142.864,A -85,B 0,C 180,E1 -8829.055,E2 -8829.055} C_VEL
LIN {X 0,Y 446.523,Z 142.863,A -85,B 0,C 180,E1 -8832.729,E2 -8832.729} C_VEL
LIN {X 0,Y 446.49,Z 142.866,A -85,B 0,C 180,E1 -8836.459,E2 -8836.459} C_VEL
LIN {X 0,Y 446.469,Z 142.873,A -85,B 0,C 180,E1 -8839.303,E2 -8839.303} C_VEL
LIN {X 0,Y 446.418,Z 142.871,A -85,B 0,C 180,E1 -8842.199,E2 -8842.199} C_VEL
LIN {X 0,Y 446.439,Z 142.875,A -85,B 0,C 180,E1 -8845.153,E2 -8845.153} C_VEL
LIN {X 0,Y 446.485,Z 142.867,A -85,B 0,C 180,E1 -8848.178,E2 -8848.178} C_VEL
LIN {X 0,Y 446.418,Z 142.875,A -85,B 0,C 180,E1 -8851.774,E2 -8851.774} C_VEL
LIN {X 0,Y 446.422,Z 142.879,A -85,B 0,C 180,E1 -8854.523,E2 -8854.523} C_VEL
LIN {X 0,Y 446.414,Z 142.882,A -85,B 0,C 180,E1 -8858.079,E2 -8858.079} C_VEL
LIN {X 0,Y 446.425,Z 142.879,A -85,B 0,C 180,E1 -8860.917,E2 -8860.917} C_VEL
LIN {X 0,Y 446.4,Z 142.883,A -85,B 0,C 180,E1 -8863.845,E2 -8863.845} C_VEL
LIN {X 0,Y 446.398,Z 142.882,A -85,B 0,C 180,E1 -8866.403,E2 -8866.403} C_VEL
LIN {X 0,Y 446.512,Z 143.028,A -85,B 0,C 180,E1 -8868.252,E2 -8868.252} C_VEL
LIN {X 0,Y 448.084,Z 151.686,A -85,B 0,C 180,E1 -8870.222,E2 -8870.222} C_VEL
LIN {X 0,Y 447.902,Z 160.357,A -85,B 0,C 180,E1 -8872.062,E2 -8872.062} C_VEL
LIN {X 0,Y 451.464,Z 177.357,A -85,B 0,C 180,E1 -8872.513,E2 -8872.513} C_VEL
LIN {X 0,Y 450.429,Z 267.688,A -85,B 0,C 180,E1 -8874.003,E2 -8874.003} C_VEL
LIN {X 0,Y 450.139,Z 280.458,A -85,B 0,C 180,E1 -8874.389,E2 -8874.389} C_VEL
LIN {X 0,Y 449.7,Z 292.956,A -85,B 0,C 180,E1 -8874.947,E2 -8874.947} C_VEL
LIN {X 0,Y 449.209,Z 303.654,A -85,B 0,C 180,E1 -8875.585,E2 -8875.585} C_VEL
LIN {X 0,Y 448.614,Z 314.858,A -85,B 0,C 180,E1 -8876.44,E2 -8876.44} C_VEL
LIN {X 0,Y 447.935,Z 325.794,A -85,B 0,C 180,E1 -8877.495,E2 -8877.495} C_VEL
LIN {X 0,Y 447.426,Z 334.499,A -85,B 0,C 180,E1 -8878.53,E2 -8878.53} C_VEL
LIN {X 0,Y 446.849,Z 343.167,A -85,B 0,C 180,E1 -8879.782,E2 -8879.782} C_VEL
LIN {X 0,Y 446.422,Z 350.257,A -85,B 0,C 180,E1 -8881.047,E2 -8881.047} C_VEL
LIN {X 0,Y 446.074,Z 356.197,A -85,B 0,C 180,E1 -8882.351,E2 -8882.351} C_VEL
LIN {X 0,Y 445.757,Z 361.998,A -85,B 0,C 180,E1 -8883.985,E2 -8883.985} C_VEL
LIN {X 0,Y 445.556,Z 365.769,A -85,B 0,C 180,E1 -8885.411,E2 -8885.411} C_VEL
LIN {X 0,Y 444.82,Z 367.332,A -85,B 0,C 180,E1 -8886.139,E2 -8886.139} C_VEL
LIN {X 0,Y 441.835,Z 369.32,A -85,B 0,C 180,E1 -8887.334,E2 -8887.334} C_VEL
LIN {X 0,Y 439.346,Z 370.412,A -85,B 0,C 180,E1 -8888.309,E2 -8888.309} C_VEL
LIN {X 0,Y 438.288,Z 370.893,A -85,B 0,C 180,E1 -8889.068,E2 -8889.068} C_VEL
LIN {X 0,Y 438.206,Z 370.978,A -85,B 0,C 180,E1 -8889.326,E2 -8889.326} C_VEL
LIN {X 0,Y 438.214,Z 370.708,A -85,B 0,C 180,E1 -8891.124,E2 -8891.124} C_VEL
LIN {X 0,Y 438.235,Z 369.778,A -85,B 0,C 180,E1 -8892.26,E2 -8892.26} C_VEL
LIN {X 0,Y 438.307,Z 368.473,A -85,B 0,C 180,E1 -8893.225,E2 -8893.225} C_VEL
LIN {X 0,Y 438.474,Z 365.691,A -85,B 0,C 180,E1 -8894.665,E2 -8894.665} C_VEL
LIN {X 0,Y 438.654,Z 361.842,A -85,B 0,C 180,E1 -8896.094,E2 -8896.094} C_VEL
LIN {X 0,Y 438.917,Z 356.438,A -85,B 0,C 180,E1 -8897.615,E2 -8897.615} C_VEL
LIN {X 0,Y 439.253,Z 350.505,A -85,B 0,C 180,E1 -8898.931,E2 -8898.931} C_VEL
LIN {X 0,Y 439.696,Z 342.6,A -85,B 0,C 180,E1 -8900.338,E2 -8900.338} C_VEL
LIN {X 0,Y 440.188,Z 334.328,A -85,B 0,C 180,E1 -8901.531,E2 -8901.531} C_VEL
LIN {X 0,Y 440.781,Z 324.63,A -85,B 0,C 180,E1 -8902.672,E2 -8902.672} C_VEL
LIN {X 0,Y 441.389,Z 313.608,A -85,B 0,C 180,E1 -8903.716,E2 -8903.716} C_VEL
LIN {X 0,Y 441.909,Z 302.801,A -85,B 0,C 180,E1 -8904.524,E2 -8904.524} C_VEL
LIN {X 0,Y 442.352,Z 290.954,A -85,B 0,C 180,E1 -8905.215,E2 -8905.215} C_VEL
LIN {X 0,Y 442.743,Z 278.174,A -85,B 0,C 180,E1 -8905.761,E2 -8905.761} C_VEL
LIN {X 0,Y 443.013,Z 265.762,A -85,B 0,C 180,E1 -8906.106,E2 -8906.106} C_VEL
LIN {X 0,Y 443.901,Z 177.239,A -85,B 0,C 180,E1 -8907.566,E2 -8907.566} C_VEL
LIN {X 0,Y 440.585,Z 160.271,A -85,B 0,C 180,E1 -8907.992,E2 -8907.992} C_VEL
LIN {X 0,Y 440.788,Z 150.942,A -85,B 0,C 180,E1 -8910,E2 -8910} C_VEL
LIN {X 0,Y 439.609,Z 143.728,A -85,B 0,C 180,E1 -8911.661,E2 -8911.661} C_VEL
LIN {X 0,Y 439.372,Z 143.761,A -85,B 0,C 180,E1 -8913.669,E2 -8913.669} C_VEL
LIN {X 0,Y 439.59,Z 143.726,A -85,B 0,C 180,E1 -8915.505,E2 -8915.505} C_VEL
LIN {X 0,Y 439.475,Z 143.741,A -85,B 0,C 180,E1 -8918.275,E2 -8918.275} C_VEL
LIN {X 0,Y 439.471,Z 143.743,A -85,B 0,C 180,E1 -8921.999,E2 -8921.999} C_VEL
LIN {X 0,Y 439.373,Z 143.751,A -85,B 0,C 180,E1 -8924.829,E2 -8924.829} C_VEL
LIN {X 0,Y 439.347,Z 143.761,A -85,B 0,C 180,E1 -8927.694,E2 -8927.694} C_VEL
LIN {X 0,Y 439.341,Z 143.754,A -85,B 0,C 180,E1 -8930.606,E2 -8930.606} C_VEL
LIN {X 0,Y 439.346,Z 143.761,A -85,B 0,C 180,E1 -8933.573,E2 -8933.573} C_VEL
LIN {X 0,Y 439.351,Z 143.754,A -85,B 0,C 180,E1 -8936.609,E2 -8936.609} C_VEL
LIN {X 0,Y 439.353,Z 143.756,A -85,B 0,C 180,E1 -8939.728,E2 -8939.728} C_VEL
LIN {X 0,Y 439.338,Z 143.759,A -85,B 0,C 180,E1 -8942.949,E2 -8942.949} C_VEL
LIN {X 0,Y 439.361,Z 143.752,A -85,B 0,C 180,E1 -8946.289,E2 -8946.289} C_VEL
LIN {X 0,Y 439.357,Z 143.753,A -85,B 0,C 180,E1 -8949.781,E2 -8949.781} C_VEL
LIN {X 0,Y 439.327,Z 143.759,A -85,B 0,C 180,E1 -8952.62,E2 -8952.62} C_VEL
LIN {X 0,Y 439.395,Z 143.751,A -85,B 0,C 180,E1 -8955.271,E2 -8955.271} C_VEL
LIN {X 0,Y 439.353,Z 143.759,A -85,B 0,C 180,E1 -8959.017,E2 -8959.017} C_VEL
LIN {X 0,Y 439.355,Z 143.753,A -85,B 0,C 180,E1 -8961.612,E2 -8961.612} C_VEL
LIN {X 0,Y 439.389,Z 143.755,A -85,B 0,C 180,E1 -8964.844,E2 -8964.844} C_VEL
LIN {X 0,Y 439.346,Z 143.756,A -85,B 0,C 180,E1 -8968.138,E2 -8968.138} C_VEL
LIN {X 0,Y 439.386,Z 143.749,A -85,B 0,C 180,E1 -8971.611,E2 -8971.611} C_VEL
LIN {X 0,Y 439.352,Z 143.76,A -85,B 0,C 180,E1 -8974.412,E2 -8974.412} C_VEL
LIN {X 0,Y 439.352,Z 143.753,A -85,B 0,C 180,E1 -8977.424,E2 -8977.424} C_VEL
LIN {X 0,Y 439.383,Z 143.752,A -85,B 0,C 180,E1 -8980.687,E2 -8980.687} C_VEL
LIN {X 0,Y 439.404,Z 143.755,A -85,B 0,C 180,E1 -8984.223,E2 -8984.223} C_VEL
LIN {X 0,Y 439.469,Z 143.739,A -85,B 0,C 180,E1 -8987.297,E2 -8987.297} C_VEL
LIN {X 0,Y 439.476,Z 143.738,A -85,B 0,C 180,E1 -8990.798,E2 -8990.798} C_VEL
LIN {X 0,Y 439.562,Z 143.73,A -85,B 0,C 180,E1 -8993.574,E2 -8993.574} C_VEL
LIN {X 0,Y 439.406,Z 143.748,A -85,B 0,C 180,E1 -8995.414,E2 -8995.414} C_VEL
LIN {X 0,Y 439.63,Z 143.723,A -85,B 0,C 180,E1 -8998.168,E2 -8998.168} C_VEL
LIN {X 0,Y 439.673,Z 143.719,A -85,B 0,C 180,E1 -9000,E2 -9000} C_VEL
LIN {X 0,Y 439.607,Z 143.721,A -85,B 0,C 180,E1 -9002.75,E2 -9002.75} C_VEL
LIN {X 0,Y 439.558,Z 143.728,A -85,B 0,C 180,E1 -9006.427,E2 -9006.427} C_VEL
LIN {X 0,Y 439.484,Z 143.74,A -85,B 0,C 180,E1 -9009.202,E2 -9009.202} C_VEL
LIN {X 0,Y 439.47,Z 143.74,A -85,B 0,C 180,E1 -9012.938,E2 -9012.938} C_VEL
LIN {X 0,Y 439.407,Z 143.746,A -85,B 0,C 180,E1 -9016.328,E2 -9016.328} C_VEL
LIN {X 0,Y 439.404,Z 143.751,A -85,B 0,C 180,E1 -9019.627,E2 -9019.627} C_VEL
LIN {X 0,Y 439.365,Z 143.752,A -85,B 0,C 180,E1 -9022.576,E2 -9022.576} C_VEL
LIN {X 0,Y 439.37,Z 143.754,A -85,B 0,C 180,E1 -9025.588,E2 -9025.588} C_VEL
LIN {X 0,Y 439.385,Z 143.752,A -85,B 0,C 180,E1 -9028.676,E2 -9028.676} C_VEL
LIN {X 0,Y 439.357,Z 143.753,A -85,B 0,C 180,E1 -9032.026,E2 -9032.026} C_VEL
LIN {X 0,Y 439.395,Z 143.751,A -85,B 0,C 180,E1 -9035.34,E2 -9035.34} C_VEL
LIN {X 0,Y 439.372,Z 143.755,A -85,B 0,C 180,E1 -9038.597,E2 -9038.597} C_VEL
LIN {X 0,Y 439.367,Z 143.754,A -85,B 0,C 180,E1 -9041.253,E2 -9041.253} C_VEL
LIN {X 0,Y 439.401,Z 143.755,A -85,B 0,C 180,E1 -9044.73,E2 -9044.73} C_VEL
LIN {X 0,Y 439.353,Z 143.753,A -85,B 0,C 180,E1 -9047.79,E2 -9047.79} C_VEL
LIN {X 0,Y 439.366,Z 143.752,A -85,B 0,C 180,E1 -9051.403,E2 -9051.403} C_VEL
LIN {X 0,Y 439.399,Z 143.75,A -85,B 0,C 180,E1 -9054.843,E2 -9054.843} C_VEL
LIN {X 0,Y 439.373,Z 143.755,A -85,B 0,C 180,E1 -9058.139,E2 -9058.139} C_VEL
LIN {X 0,Y 439.403,Z 143.751,A -85,B 0,C 180,E1 -9061.606,E2 -9061.606} C_VEL
LIN {X 0,Y 439.41,Z 143.852,A -85,B 0,C 180,E1 -9063.298,E2 -9063.298} C_VEL
LIN {X 0,Y 441.852,Z 156.497,A -85,B 0,C 180,E1 -9065.822,E2 -9065.822} C_VEL
LIN {X 0,Y 441.517,Z 165.763,A -85,B 0,C 180,E1 -9067.54,E2 -9067.54} C_VEL
LIN {X 0,Y 440.542,Z 185.501,A -85,B 0,C 180,E1 -9071.152,E2 -9071.152} C_VEL
LIN {X 0,Y 440.342,Z 190.609,A -85,B 0,C 180,E1 -9072.038,E2 -9072.038} C_VEL
LIN {X 0,Y 443.638,Z 213.289,A -85,B 0,C 180,E1 -9072.539,E2 -9072.539} C_VEL
LIN {X 0,Y 442.835,Z 298.981,A -85,B 0,C 180,E1 -9073.963,E2 -9073.963} C_VEL
LIN {X 0,Y 442.408,Z 312.17,A -85,B 0,C 180,E1 -9074.362,E2 -9074.362} C_VEL
LIN {X 0,Y 441.932,Z 324.32,A -85,B 0,C 180,E1 -9074.905,E2 -9074.905} C_VEL
LIN {X 0,Y 441.367,Z 335.779,A -85,B 0,C 180,E1 -9075.593,E2 -9075.593} C_VEL
LIN {X 0,Y 440.714,Z 347.517,A -85,B 0,C 180,E1 -9076.509,E2 -9076.509} C_VEL
LIN {X 0,Y 440.11,Z 358.132,A -85,B 0,C 180,E1 -9077.55,E2 -9077.55} C_VEL
LIN {X 0,Y 439.649,Z 367.662,A -85,B 0,C 180,E1 -9078.707,E2 -9078.707} C_VEL
LIN {X 0,Y 439.102,Z 376.822,A -85,B 0,C 180,E1 -9080.092,E2 -9080.092} C_VEL
LIN {X 0,Y 438.727,Z 384.2,A -85,B 0,C 180,E1 -9081.479,E2 -9081.479} C_VEL
LIN {X 0,Y 438.529,Z 389.198,A -85,B 0,C 180,E1 -9082.634,E2 -9082.634} C_VEL
LIN {X 0,Y 438.346,Z 394.067,A -85,B 0,C 180,E1 -9084.026,E2 -9084.026} C_VEL
LIN {X 0,Y 438.34,Z 397.754,A -85,B 0,C 180,E1 -9085.402,E2 -9085.402} C_VEL
LIN {X 0,Y 438.284,Z 399.667,A -85,B 0,C 180,E1 -9086.322,E2 -9086.322} C_VEL
LIN {X 0,Y 438.342,Z 401.137,A -85,B 0,C 180,E1 -9087.243,E2 -9087.243} C_VEL
LIN {X 0,Y 438.281,Z 402.806,A -85,B 0,C 180,E1 -9089.081,E2 -9089.081} C_VEL
LIN {X 0,Y 438.284,Z 403.057,A -85,B 0,C 180,E1 -9090,E2 -9090} C_VEL
LIN {X 0,Y 438.257,Z 402.893,A -85,B 0,C 180,E1 -9090.919,E2 -9090.919} C_VEL
LIN {X 0,Y 438.296,Z 402.31,A -85,B 0,C 180,E1 -9091.838,E2 -9091.838} C_VEL
LIN {X 0,Y 438.341,Z 401.337,A -85,B 0,C 180,E1 -9092.757,E2 -9092.757} C_VEL
LIN {X 0,Y 438.281,Z 399.966,A -85,B 0,C 180,E1 -9093.677,E2 -9093.677} C_VEL
LIN {X 0,Y 438.379,Z 397.079,A -85,B 0,C 180,E1 -9095.058,E2 -9095.058} C_VEL
LIN {X 0,Y 438.372,Z 393.161,A -85,B 0,C 180,E1 -9096.443,E2 -9096.443} C_VEL
LIN {X 0,Y 438.639,Z 388.123,A -85,B 0,C 180,E1 -9097.827,E2 -9097.827} C_VEL
LIN {X 0,Y 438.948,Z 381.805,A -85,B 0,C 180,E1 -9099.213,E2 -9099.213} C_VEL
LIN {X 0,Y 439.341,Z 373.908,A -85,B 0,C 180,E1 -9100.601,E2 -9100.601} C_VEL
LIN {X 0,Y 440.051,Z 364.091,A -85,B 0,C 180,E1 -9101.983,E2 -9101.983} C_VEL
LIN {X 0,Y 440.63,Z 354.538,A -85,B 0,C 180,E1 -9103.072,E2 -9103.072} C_VEL
LIN {X 0,Y 441.277,Z 343.814,A -85,B 0,C 180,E1 -9104.056,E2 -9104.056} C_VEL
LIN {X 0,Y 441.952,Z 332.85,A -85,B 0,C 180,E1 -9104.858,E2 -9104.858} C_VEL
LIN {X 0,Y 442.66,Z 320.736,A -85,B 0,C 180,E1 -9105.54,E2 -9105.54} C_VEL
LIN {X 0,Y 443.132,Z 308.208,A -85,B 0,C 180,E1 -9106.055,E2 -9106.055} C_VEL
LIN {X 0,Y 443.649,Z 295.151,A -85,B 0,C 180,E1 -9106.39,E2 -9106.39} C_VEL
LIN {X 0,Y 444.272,Z 212.865,A -85,B 0,C 180,E1 -9107.767,E2 -9107.767} C_VEL
LIN {X 0,Y 440.715,Z 190.925,A -85,B 0,C 180,E1 -9108.307,E2 -9108.307} C_VEL
LIN {X 0,Y 440.569,Z 189.697,A -85,B 0,C 180,E1 -9108.369,E2 -9108.369} C_VEL
LIN {X 0,Y 441.585,Z 171.542,A -85,B 0,C 180,E1 -9111.718,E2 -9111.718} C_VEL
LIN {X 0,Y 442.278,Z 158.581,A -85,B 0,C 180,E1 -9114.153,E2 -9114.153} C_VEL
LIN {X 0,Y 440.255,Z 147.67,A -85,B 0,C 180,E1 -9116.398,E2 -9116.398} C_VEL
LIN {X 0,Y 439.4,Z 143.754,A -85,B 0,C 180,E1 -9117.248,E2 -9117.248} C_VEL
LIN {X 0,Y 439.382,Z 143.756,A -85,B 0,C 180,E1 -9120.26,E2 -9120.26} C_VEL
LIN {X 0,Y 439.366,Z 143.754,A -85,B 0,C 180,E1 -9123.717,E2 -9123.717} C_VEL
LIN {X 0,Y 439.373,Z 143.753,A -85,B 0,C 180,E1 -9126.287,E2 -9126.287} C_VEL
LIN {X 0,Y 439.361,Z 143.754,A -85,B 0,C 180,E1 -9129.78,E2 -9129.78} C_VEL
LIN {X 0,Y 439.335,Z 143.759,A -85,B 0,C 180,E1 -9132.62,E2 -9132.62} C_VEL
LIN {X 0,Y 439.399,Z 143.754,A -85,B 0,C 180,E1 -9135.27,E2 -9135.27} C_VEL
LIN {X 0,Y 439.353,Z 143.757,A -85,B 0,C 180,E1 -9139.016,E2 -9139.016} C_VEL
LIN {X 0,Y 439.354,Z 143.753,A -85,B 0,C 180,E1 -9141.611,E2 -9141.611} C_VEL
LIN {X 0,Y 439.387,Z 143.752,A -85,B 0,C 180,E1 -9144.842,E2 -9144.842} C_VEL
LIN {X 0,Y 439.347,Z 143.756,A -85,B 0,C 180,E1 -9148.137,E2 -9148.137} C_VEL
LIN {X 0,Y 439.379,Z 143.75,A -85,B 0,C 180,E1 -9151.323,E2 -9151.323} C_VEL
LIN {X 0,Y 439.356,Z 143.755,A -85,B 0,C 180,E1 -9154.412,E2 -9154.412} C_VEL
LIN {X 0,Y 439.354,Z 143.747,A -85,B 0,C 180,E1 -9157.423,E2 -9157.423} C_VEL
LIN {X 0,Y 439.383,Z 143.75,A -85,B 0,C 180,E1 -9160.686,E2 -9160.686} C_VEL
LIN {X 0,Y 439.419,Z 143.753,A -85,B 0,C 180,E1 -9164.222,E2 -9164.222} C_VEL
LIN {X 0,Y 439.487,Z 143.73,A -85,B 0,C 180,E1 -9167.285,E2 -9167.285} C_VEL
LIN {X 0,Y 439.485,Z 143.734,A -85,B 0,C 180,E1 -9170.798,E2 -9170.798} C_VEL
LIN {X 0,Y 439.562,Z 143.729,A -85,B 0,C 180,E1 -9173.573,E2 -9173.573} C_VEL
LIN {X 0,Y 439.41,Z 143.749,A -85,B 0,C 180,E1 -9175.413,E2 -9175.413} C_VEL
LIN {X 0,Y 439.629,Z 143.721,A -85,B 0,C 180,E1 -9178.167,E2 -9178.167} C_VEL
LIN {X 0,Y 439.713,Z 143.708,A -85,B 0,C 180,E1 -9180,E2 -9180} C_VEL
LIN {X 0,Y 439.633,Z 143.717,A -85,B 0,C 180,E1 -9182.748,E2 -9182.748} C_VEL
LIN {X 0,Y 439.567,Z 143.723,A -85,B 0,C 180,E1 -9186.425,E2 -9186.425} C_VEL
LIN {X 0,Y 439.497,Z 143.741,A -85,B 0,C 180,E1 -9189.201,E2 -9189.201} C_VEL
LIN {X 0,Y 439.467,Z 143.744,A -85,B 0,C 180,E1 -9192.937,E2 -9192.937} C_VEL
LIN {X 0,Y 439.448,Z 143.743,A -85,B 0,C 180,E1 -9196.347,E2 -9196.347} C_VEL
LIN {X 0,Y 439.403,Z 143.75,A -85,B 0,C 180,E1 -9199.626,E2 -9199.626} C_VEL
LIN {X 0,Y 439.364,Z 143.753,A -85,B 0,C 180,E1 -9202.575,E2 -9202.575} C_VEL
LIN {X 0,Y 439.387,Z 143.751,A -85,B 0,C 180,E1 -9205.585,E2 -9205.585} C_VEL
LIN {X 0,Y 439.417,Z 143.751,A -85,B 0,C 180,E1 -9208.673,E2 -9208.673} C_VEL
LIN {X 0,Y 439.368,Z 143.755,A -85,B 0,C 180,E1 -9212.029,E2 -9212.029} C_VEL
LIN {X 0,Y 439.391,Z 143.752,A -85,B 0,C 180,E1 -9215.339,E2 -9215.339} C_VEL
LIN {X 0,Y 439.377,Z 143.754,A -85,B 0,C 180,E1 -9218.595,E2 -9218.595} C_VEL
LIN {X 0,Y 439.387,Z 143.755,A -85,B 0,C 180,E1 -9221.256,E2 -9221.256} C_VEL
LIN {X 0,Y 439.4,Z 143.754,A -85,B 0,C 180,E1 -9224.729,E2 -9224.729} C_VEL
LIN {X 0,Y 439.432,Z 143.838,A -85,B 0,C 180,E1 -9227.97,E2 -9227.97} C_VEL
LIN {X 0,Y 441.059,Z 152.105,A -85,B 0,C 180,E1 -9229.893,E2 -9229.893} C_VEL
LIN {X 0,Y 441.144,Z 158.615,A -85,B 0,C 180,E1 -9231.318,E2 -9231.318} C_VEL
LIN {X 0,Y 441.037,Z 160.497,A -85,B 0,C 180,E1 -9231.72,E2 -9231.72} C_VEL
LIN {X 0,Y 444.802,Z 178.5,A -85,B 0,C 180,E1 -9232.227,E2 -9232.227} C_VEL
LIN {X 0,Y 443.688,Z 267.947,A -85,B 0,C 180,E1 -9233.724,E2 -9233.724} C_VEL
LIN {X 0,Y 443.365,Z 280.982,A -85,B 0,C 180,E1 -9234.125,E2 -9234.125} C_VEL
LIN {X 0,Y 442.843,Z 294.371,A -85,B 0,C 180,E1 -9234.741,E2 -9234.741} C_VEL
LIN {X 0,Y 442.289,Z 306.326,A -85,B 0,C 180,E1 -9235.501,E2 -9235.501} C_VEL
LIN {X 0,Y 441.635,Z 317.675,A -85,B 0,C 180,E1 -9236.427,E2 -9236.427} C_VEL
LIN {X 0,Y 440.943,Z 328.044,A -85,B 0,C 180,E1 -9237.486,E2 -9237.486} C_VEL
LIN {X 0,Y 440.272,Z 337.896,A -85,B 0,C 180,E1 -9238.749,E2 -9238.749} C_VEL
LIN {X 0,Y 439.757,Z 345.606,A -85,B 0,C 180,E1 -9239.961,E2 -9239.961} C_VEL
LIN {X 0,Y 439.262,Z 352.64,A -85,B 0,C 180,E1 -9241.315,E2 -9241.315} C_VEL
LIN {X 0,Y 438.895,Z 358.937,A -85,B 0,C 180,E1 -9242.847,E2 -9242.847} C_VEL
LIN {X 0,Y 438.621,Z 363.717,A -85,B 0,C 180,E1 -9244.366,E2 -9244.366} C_VEL
LIN {X 0,Y 438.41,Z 367.503,A -85,B 0,C 180,E1 -9246.027,E2 -9246.027} C_VEL
LIN {X 0,Y 438.29,Z 369.534,A -85,B 0,C 180,E1 -9247.366,E2 -9247.366} C_VEL
LIN {X 0,Y 438.247,Z 370.577,A -85,B 0,C 180,E1 -9248.452,E2 -9248.452} C_VEL
LIN {X 0,Y 438.206,Z 370.978,A -85,B 0,C 180,E1 -9249.326,E2 -9249.326} C_VEL
LIN {X 0,Y 437.542,Z 371.174,A -85,B 0,C 180,E1 -9250.093,E2 -9250.093} C_VEL
LIN {X 0,Y 434.671,Z 370.824,A -85,B 0,C 180,E1 -9251.34,E2 -9251.34} C_VEL
LIN {X 0,Y 432.271,Z 369.936,A -85,B 0,C 180,E1 -9252.341,E2 -9252.341} C_VEL
LIN {X 0,Y 431.285,Z 368.945,A -85,B 0,C 180,E1 -9253.108,E2 -9253.108} C_VEL
LIN {X 0,Y 431.23,Z 368.502,A -85,B 0,C 180,E1 -9253.366,E2 -9253.366} C_VEL
LIN {X 0,Y 431.434,Z 365.535,A -85,B 0,C 180,E1 -9254.892,E2 -9254.892} C_VEL
LIN {X 0,Y 431.607,Z 361.553,A -85,B 0,C 180,E1 -9256.343,E2 -9256.343} C_VEL
LIN {X 0,Y 431.895,Z 356.389,A -85,B 0,C 180,E1 -9257.787,E2 -9257.787} C_VEL
LIN {X 0,Y 432.258,Z 349.874,A -85,B 0,C 180,E1 -9259.224,E2 -9259.224} C_VEL
LIN {X 0,Y 432.725,Z 341.735,A -85,B 0,C 180,E1 -9260.653,E2 -9260.653} C_VEL
LIN {X 0,Y 433.31,Z 332.924,A -85,B 0,C 180,E1 -9261.905,E2 -9261.905} C_VEL
LIN {X 0,Y 433.907,Z 323.247,A -85,B 0,C 180,E1 -9263.023,E2 -9263.023} C_VEL
LIN {X 0,Y 434.578,Z 311.703,A -85,B 0,C 180,E1 -9264.083,E2 -9264.083} C_VEL
LIN {X 0,Y 435.104,Z 300.404,A -85,B 0,C 180,E1 -9264.903,E2 -9264.903} C_VEL
LIN {X 0,Y 435.543,Z 288.926,A -85,B 0,C 180,E1 -9265.546,E2 -9265.546} C_VEL
LIN {X 0,Y 435.876,Z 275.825,A -85,B 0,C 180,E1 -9266.071,E2 -9266.071} C_VEL
LIN {X 0,Y 436.221,Z 262.174,A -85,B 0,C 180,E1 -9266.408,E2 -9266.408} C_VEL
LIN {X 0,Y 437.026,Z 178.066,A -85,B 0,C 180,E1 -9267.81,E2 -9267.81} C_VEL
LIN {X 0,Y 433.636,Z 160.487,A -85,B 0,C 180,E1 -9268.259,E2 -9268.259} C_VEL
LIN {X 0,Y 433.853,Z 152.491,A -85,B 0,C 180,E1 -9270,E2 -9270} C_VEL
LIN {X 0,Y 432.597,Z 144.602,A -85,B 0,C 180,E1 -9271.833,E2 -9271.833} C_VEL
LIN {X 0,Y 432.545,Z 144.604,A -85,B 0,C 180,E1 -9275.595,E2 -9275.595} C_VEL
LIN {X 0,Y 432.442,Z 144.616,A -85,B 0,C 180,E1 -9278.411,E2 -9278.411} C_VEL
LIN {X 0,Y 432.445,Z 144.616,A -85,B 0,C 180,E1 -9282.197,E2 -9282.197} C_VEL
LIN {X 0,Y 432.352,Z 144.628,A -85,B 0,C 180,E1 -9286.042,E2 -9286.042} C_VEL
LIN {X 0,Y 432.338,Z 144.633,A -85,B 0,C 180,E1 -9289.469,E2 -9289.469} C_VEL
LIN {X 0,Y 432.331,Z 144.629,A -85,B 0,C 180,E1 -9292.092,E2 -9292.092} C_VEL
LIN {X 0,Y 432.308,Z 144.633,A -85,B 0,C 180,E1 -9295.004,E2 -9295.004} C_VEL
LIN {X 0,Y 432.308,Z 144.631,A -85,B 0,C 180,E1 -9298.129,E2 -9298.129} C_VEL
LIN {X 0,Y 432.296,Z 144.639,A -85,B 0,C 180,E1 -9301.349,E2 -9301.349} C_VEL
LIN {X 0,Y 432.319,Z 144.631,A -85,B 0,C 180,E1 -9304.679,E2 -9304.679} C_VEL
LIN {X 0,Y 432.316,Z 144.63,A -85,B 0,C 180,E1 -9308.153,E2 -9308.153} C_VEL
LIN {X 0,Y 432.299,Z 144.632,A -85,B 0,C 180,E1 -9311.802,E2 -9311.802} C_VEL
LIN {X 0,Y 432.332,Z 144.629,A -85,B 0,C 180,E1 -9314.348,E2 -9314.348} C_VEL
LIN {X 0,Y 432.299,Z 144.638,A -85,B 0,C 180,E1 -9317.019,E2 -9317.019} C_VEL
LIN {X 0,Y 432.287,Z 144.633,A -85,B 0,C 180,E1 -9319.829,E2 -9319.829} C_VEL
LIN {X 0,Y 432.296,Z 144.636,A -85,B 0,C 180,E1 -9323.022,E2 -9323.022} C_VEL
LIN {X 0,Y 432.33,Z 144.629,A -85,B 0,C 180,E1 -9326.003,E2 -9326.003} C_VEL
LIN {X 0,Y 432.331,Z 144.628,A -85,B 0,C 180,E1 -9329.494,E2 -9329.494} C_VEL
LIN {X 0,Y 432.313,Z 144.631,A -85,B 0,C 180,E1 -9331.872,E2 -9331.872} C_VEL
LIN {X 0,Y 432.314,Z 144.632,A -85,B 0,C 180,E1 -9334.997,E2 -9334.997} C_VEL
LIN {X 0,Y 432.351,Z 144.629,A -85,B 0,C 180,E1 -9338.046,E2 -9338.046} C_VEL
LIN {X 0,Y 432.339,Z 144.627,A -85,B 0,C 180,E1 -9341.028,E2 -9341.028} C_VEL
LIN {X 0,Y 432.359,Z 144.628,A -85,B 0,C 180,E1 -9343.959,E2 -9343.959} C_VEL
LIN {X 0,Y 432.453,Z 144.616,A -85,B 0,C 180,E1 -9347.804,E2 -9347.804} C_VEL
LIN {X 0,Y 432.449,Z 144.615,A -85,B 0,C 180,E1 -9351.59,E2 -9351.59} C_VEL
LIN {X 0,Y 432.554,Z 144.602,A -85,B 0,C 180,E1 -9354.406,E2 -9354.406} C_VEL
LIN {X 0,Y 432.599,Z 144.599,A -85,B 0,C 180,E1 -9358.139,E2 -9358.139} C_VEL
LIN {X 0,Y 432.625,Z 144.597,A -85,B 0,C 180,E1 -9360.001,E2 -9360.001} C_VEL
LIN {X 0,Y 432.56,Z 144.599,A -85,B 0,C 180,E1 -9362.794,E2 -9362.794} C_VEL
LIN {X 0,Y 432.515,Z 144.605,A -85,B 0,C 180,E1 -9366.532,E2 -9366.532} C_VEL
LIN {X 0,Y 432.43,Z 144.62,A -85,B 0,C 180,E1 -9369.354,E2 -9369.354} C_VEL
LIN {X 0,Y 432.436,Z 144.615,A -85,B 0,C 180,E1 -9372.803,E2 -9372.803} C_VEL
LIN {X 0,Y 432.366,Z 144.623,A -85,B 0,C 180,E1 -9376.455,E2 -9376.455} C_VEL
LIN {X 0,Y 432.391,Z 144.626,A -85,B 0,C 180,E1 -9379.485,E2 -9379.485} C_VEL
LIN {X 0,Y 432.313,Z 144.634,A -85,B 0,C 180,E1 -9382.965,E2 -9382.965} C_VEL
LIN {X 0,Y 432.322,Z 144.629,A -85,B 0,C 180,E1 -9386.036,E2 -9386.036} C_VEL
LIN {X 0,Y 432.326,Z 144.635,A -85,B 0,C 180,E1 -9389.189,E2 -9389.189} C_VEL
LIN {X 0,Y 432.32,Z 144.63,A -85,B 0,C 180,E1 -9392.444,E2 -9392.444} C_VEL
LIN {X 0,Y 432.341,Z 144.627,A -85,B 0,C 180,E1 -9395.818,E2 -9395.818} C_VEL
LIN {X 0,Y 432.334,Z 144.633,A -85,B 0,C 180,E1 -9398.712,E2 -9398.712} C_VEL
LIN {X 0,Y 432.308,Z 144.631,A -85,B 0,C 180,E1 -9401.801,E2 -9401.801} C_VEL
LIN {X 0,Y 432.338,Z 144.63,A -85,B 0,C 180,E1 -9404.347,E2 -9404.347} C_VEL
LIN {X 0,Y 432.306,Z 144.634,A -85,B 0,C 180,E1 -9407.018,E2 -9407.018} C_VEL
LIN {X 0,Y 432.294,Z 144.633,A -85,B 0,C 180,E1 -9409.828,E2 -9409.828} C_VEL
LIN {X 0,Y 432.308,Z 144.632,A -85,B 0,C 180,E1 -9413.022,E2 -9413.022} C_VEL
LIN {X 0,Y 432.337,Z 144.63,A -85,B 0,C 180,E1 -9416.002,E2 -9416.002} C_VEL
LIN {X 0,Y 432.35,Z 144.629,A -85,B 0,C 180,E1 -9419.49,E2 -9419.49} C_VEL
LIN {X 0,Y 432.36,Z 144.633,A -85,B 0,C 180,E1 -9422.926,E2 -9422.926} C_VEL
LIN {X 0,Y 432.403,Z 144.886,A -85,B 0,C 180,E1 -9423.126,E2 -9423.126} C_VEL
LIN {X 0,Y 434.841,Z 157.351,A -85,B 0,C 180,E1 -9425.66,E2 -9425.66} C_VEL
LIN {X 0,Y 434.715,Z 163.981,A -85,B 0,C 180,E1 -9426.918,E2 -9426.918} C_VEL
LIN {X 0,Y 433.721,Z 182.445,A -85,B 0,C 180,E1 -9430.352,E2 -9430.352} C_VEL
LIN {X 0,Y 433.343,Z 190.095,A -85,B 0,C 180,E1 -9431.764,E2 -9431.764} C_VEL
LIN {X 0,Y 436.813,Z 214.527,A -85,B 0,C 180,E1 -9432.314,E2 -9432.314} C_VEL
LIN {X 0,Y 435.971,Z 298.643,A -85,B 0,C 180,E1 -9433.734,E2 -9433.734} C_VEL
LIN {X 0,Y 435.502,Z 311.853,A -85,B 0,C 180,E1 -9434.137,E2 -9434.137} C_VEL
LIN {X 0,Y 434.995,Z 324.586,A -85,B 0,C 180,E1 -9434.719,E2 -9434.719} C_VEL
LIN {X 0,Y 434.365,Z 336.697,A -85,B 0,C 180,E1 -9435.476,E2 -9435.476} C_VEL
LIN {X 0,Y 433.683,Z 348.56,A -85,B 0,C 180,E1 -9436.438,E2 -9436.438} C_VEL
LIN {X 0,Y 433.066,Z 358.662,A -85,B 0,C 180,E1 -9437.464,E2 -9437.464} C_VEL
LIN {X 0,Y 432.629,Z 367.174,A -85,B 0,C 180,E1 -9438.521,E2 -9438.521} C_VEL
LIN {X 0,Y 432.045,Z 376.38,A -85,B 0,C 180,E1 -9439.929,E2 -9439.929} C_VEL
LIN {X 0,Y 431.679,Z 383.793,A -85,B 0,C 180,E1 -9441.338,E2 -9441.338} C_VEL
LIN {X 0,Y 431.416,Z 390.59,A -85,B 0,C 180,E1 -9442.982,E2 -9442.982} C_VEL
LIN {X 0,Y 431.262,Z 395.067,A -85,B 0,C 180,E1 -9444.389,E2 -9444.389} C_VEL
LIN {X 0,Y 431.268,Z 397.429,A -85,B 0,C 180,E1 -9445.326,E2 -9445.326} C_VEL
LIN {X 0,Y 431.19,Z 399.353,A -85,B 0,C 180,E1 -9446.262,E2 -9446.262} C_VEL
LIN {X 0,Y 431.253,Z 400.844,A -85,B 0,C 180,E1 -9447.197,E2 -9447.197} C_VEL
LIN {X 0,Y 431.219,Z 401.884,A -85,B 0,C 180,E1 -9448.132,E2 -9448.132} C_VEL
LIN {X 0,Y 431.197,Z 402.792,A -85,B 0,C 180,E1 -9450,E2 -9450} C_VEL
LIN {X 0,Y 431.174,Z 402.647,A -85,B 0,C 180,E1 -9450.934,E2 -9450.934} C_VEL
LIN {X 0,Y 431.219,Z 402.074,A -85,B 0,C 180,E1 -9451.868,E2 -9451.868} C_VEL
LIN {X 0,Y 431.237,Z 401.111,A -85,B 0,C 180,E1 -9452.802,E2 -9452.802} C_VEL
LIN {X 0,Y 431.188,Z 399.749,A -85,B 0,C 180,E1 -9453.738,E2 -9453.738} C_VEL
LIN {X 0,Y 431.288,Z 396.883,A -85,B 0,C 180,E1 -9455.142,E2 -9455.142} C_VEL
LIN {X 0,Y 431.293,Z 392.986,A -85,B 0,C 180,E1 -9456.55,E2 -9456.55} C_VEL
LIN {X 0,Y 431.558,Z 387.97,A -85,B 0,C 180,E1 -9457.957,E2 -9457.957} C_VEL
LIN {X 0,Y 431.912,Z 381.68,A -85,B 0,C 180,E1 -9459.365,E2 -9459.365} C_VEL
LIN {X 0,Y 432.347,Z 373.825,A -85,B 0,C 180,E1 -9460.774,E2 -9460.774} C_VEL
LIN {X 0,Y 433.095,Z 364.043,A -85,B 0,C 180,E1 -9462.178,E2 -9462.178} C_VEL
LIN {X 0,Y 433.728,Z 353.698,A -85,B 0,C 180,E1 -9463.372,E2 -9463.372} C_VEL
LIN {X 0,Y 434.485,Z 342.468,A -85,B 0,C 180,E1 -9464.4,E2 -9464.4} C_VEL
LIN {X 0,Y 435.214,Z 331.247,A -85,B 0,C 180,E1 -9465.213,E2 -9465.213} C_VEL
LIN {X 0,Y 435.939,Z 318.645,A -85,B 0,C 180,E1 -9465.906,E2 -9465.906} C_VEL
LIN {X 0,Y 436.463,Z 306.1,A -85,B 0,C 180,E1 -9466.397,E2 -9466.397} C_VEL
LIN {X 0,Y 436.919,Z 293.372,A -85,B 0,C 180,E1 -9466.71,E2 -9466.71} C_VEL
LIN {X 0,Y 437.581,Z 213.645,A -85,B 0,C 180,E1 -9468.061,E2 -9468.061} C_VEL
LIN {X 0,Y 434.177,Z 192.547,A -85,B 0,C 180,E1 -9468.595,E2 -9468.595} C_VEL
LIN {X 0,Y 433.667,Z 189.47,A -85,B 0,C 180,E1 -9468.699,E2 -9468.699} C_VEL
LIN {X 0,Y 434.74,Z 171.5,A -85,B 0,C 180,E1 -9472.077,E2 -9472.077} C_VEL
LIN {X 0,Y 435.366,Z 159.838,A -85,B 0,C 180,E1 -9474.308,E2 -9474.308} C_VEL
LIN {X 0,Y 433.507,Z 149.84,A -85,B 0,C 180,E1 -9476.399,E2 -9476.399} C_VEL
LIN {X 0,Y 432.333,Z 144.637,A -85,B 0,C 180,E1 -9477.534,E2 -9477.534} C_VEL
LIN {X 0,Y 432.349,Z 144.633,A -85,B 0,C 180,E1 -9480.51,E2 -9480.51} C_VEL
LIN {X 0,Y 432.335,Z 144.627,A -85,B 0,C 180,E1 -9483.998,E2 -9483.998} C_VEL
LIN {X 0,Y 432.32,Z 144.63,A -85,B 0,C 180,E1 -9487.196,E2 -9487.196} C_VEL
LIN {X 0,Y 432.29,Z 144.633,A -85,B 0,C 180,E1 -9490.172,E2 -9490.172} C_VEL
LIN {X 0,Y 432.304,Z 144.639,A -85,B 0,C 180,E1 -9493.063,E2 -9493.063} C_VEL
LIN {X 0,Y 432.335,Z 144.63,A -85,B 0,C 180,E1 -9495.665,E2 -9495.665} C_VEL
LIN {X 0,Y 432.307,Z 144.634,A -85,B 0,C 180,E1 -9498.402,E2 -9498.402} C_VEL
LIN {X 0,Y 432.32,Z 144.628,A -85,B 0,C 180,E1 -9501.848,E2 -9501.848} C_VEL
LIN {X 0,Y 432.322,Z 144.628,A -85,B 0,C 180,E1 -9505.321,E2 -9505.321} C_VEL
LIN {X 0,Y 432.301,Z 144.633,A -85,B 0,C 180,E1 -9508.652,E2 -9508.652} C_VEL
LIN {X 0,Y 432.314,Z 144.631,A -85,B 0,C 180,E1 -9511.871,E2 -9511.871} C_VEL
LIN {X 0,Y 432.348,Z 144.626,A -85,B 0,C 180,E1 -9515.548,E2 -9515.548} C_VEL
LIN {X 0,Y 432.323,Z 144.63,A -85,B 0,C 180,E1 -9519.044,E2 -9519.044} C_VEL
LIN {X 0,Y 432.318,Z 144.629,A -85,B 0,C 180,E1 -9522.008,E2 -9522.008} C_VEL
LIN {X 0,Y 432.35,Z 144.627,A -85,B 0,C 180,E1 -9524.924,E2 -9524.924} C_VEL
LIN {X 0,Y 432.457,Z 144.61,A -85,B 0,C 180,E1 -9527.803,E2 -9527.803} C_VEL
LIN {X 0,Y 432.452,Z 144.612,A -85,B 0,C 180,E1 -9531.589,E2 -9531.589} C_VEL
LIN {X 0,Y 432.575,Z 144.599,A -85,B 0,C 180,E1 -9534.405,E2 -9534.405} C_VEL
LIN {X 0,Y 432.598,Z 144.597,A -85,B 0,C 180,E1 -9538.138,E2 -9538.138} C_VEL
LIN {X 0,Y 432.663,Z 144.586,A -85,B 0,C 180,E1 -9539.999,E2 -9539.999} C_VEL
LIN {X 0,Y 432.584,Z 144.595,A -85,B 0,C 180,E1 -9542.793,E2 -9542.793} C_VEL
LIN {X 0,Y 432.58,Z 144.596,A -85,B 0,C 180,E1 -9545.594,E2 -9545.594} C_VEL
LIN {X 0,Y 432.465,Z 144.612,A -85,B 0,C 180,E1 -9548.41,E2 -9548.41} C_VEL
LIN {X 0,Y 432.461,Z 144.613,A -85,B 0,C 180,E1 -9552.196,E2 -9552.196} C_VEL
LIN {X 0,Y 432.431,Z 144.617,A -85,B 0,C 180,E1 -9556.038,E2 -9556.038} C_VEL
LIN {X 0,Y 432.387,Z 144.625,A -85,B 0,C 180,E1 -9559.484,E2 -9559.484} C_VEL
LIN {X 0,Y 432.317,Z 144.636,A -85,B 0,C 180,E1 -9562.964,E2 -9562.964} C_VEL
LIN {X 0,Y 432.35,Z 144.628,A -85,B 0,C 180,E1 -9566.033,E2 -9566.033} C_VEL
LIN {X 0,Y 432.343,Z 144.631,A -85,B 0,C 180,E1 -9569.187,E2 -9569.187} C_VEL
LIN {X 0,Y 432.322,Z 144.635,A -85,B 0,C 180,E1 -9572.442,E2 -9572.442} C_VEL
LIN {X 0,Y 432.342,Z 144.63,A -85,B 0,C 180,E1 -9575.631,E2 -9575.631} C_VEL
LIN {X 0,Y 432.345,Z 144.63,A -85,B 0,C 180,E1 -9579.343,E2 -9579.343} C_VEL
LIN {X 0,Y 432.332,Z 144.634,A -85,B 0,C 180,E1 -9581.796,E2 -9581.796} C_VEL
LIN {X 0,Y 432.332,Z 144.634,A -85,B 0,C 180,E1 -9584.347,E2 -9584.347} C_VEL
LIN {X 0,Y 432.361,Z 144.661,A -85,B 0,C 180,E1 -9587.679,E2 -9587.679} C_VEL
LIN {X 0,Y 434.011,Z 152.888,A -85,B 0,C 180,E1 -9589.63,E2 -9589.63} C_VEL
LIN {X 0,Y 434.312,Z 157.056,A -85,B 0,C 180,E1 -9590.57,E2 -9590.57} C_VEL
LIN {X 0,Y 434.197,Z 160.992,A -85,B 0,C 180,E1 -9591.402,E2 -9591.402} C_VEL
LIN {X 0,Y 438.123,Z 179.236,A -85,B 0,C 180,E1 -9591.923,E2 -9591.923} C_VEL
LIN {X 0,Y 436.965,Z 268.51,A -85,B 0,C 180,E1 -9593.445,E2 -9593.445} C_VEL
LIN {X 0,Y 436.621,Z 281.605,A -85,B 0,C 180,E1 -9593.858,E2 -9593.858} C_VEL
LIN {X 0,Y 436.088,Z 294.587,A -85,B 0,C 180,E1 -9594.466,E2 -9594.466} C_VEL
LIN {X 0,Y 435.54,Z 305.526,A -85,B 0,C 180,E1 -9595.161,E2 -9595.161} C_VEL
LIN {X 0,Y 434.829,Z 317.171,A -85,B 0,C 180,E1 -9596.109,E2 -9596.109} C_VEL
LIN {X 0,Y 434.058,Z 328.308,A -85,B 0,C 180,E1 -9597.255,E2 -9597.255} C_VEL
LIN {X 0,Y 433.38,Z 337.68,A -85,B 0,C 180,E1 -9598.467,E2 -9598.467} C_VEL
LIN {X 0,Y 432.781,Z 345.903,A -85,B 0,C 180,E1 -9599.774,E2 -9599.774} C_VEL
LIN {X 0,Y 432.272,Z 352.983,A -85,B 0,C 180,E1 -9601.161,E2 -9601.161} C_VEL
LIN {X 0,Y 431.951,Z 357.994,A -85,B 0,C 180,E1 -9602.374,E2 -9602.374} C_VEL
LIN {X 0,Y 431.62,Z 363.101,A -85,B 0,C 180,E1 -9603.919,E2 -9603.919} C_VEL
LIN {X 0,Y 431.472,Z 365.727,A -85,B 0,C 180,E1 -9604.944,E2 -9604.944} C_VEL
LIN {X 0,Y 431.349,Z 367.824,A -85,B 0,C 180,E1 -9605.963,E2 -9605.963} C_VEL
LIN {X 0,Y 431.222,Z 369.42,A -85,B 0,C 180,E1 -9606.974,E2 -9606.974} C_VEL
LIN {X 0,Y 431.156,Z 370.76,A -85,B 0,C 180,E1 -9608.296,E2 -9608.296} C_VEL
LIN {X 0,Y 431.104,Z 371.328,A -85,B 0,C 180,E1 -9609.98,E2 -9609.98} C_VEL
LIN {X 0,Y 431.108,Z 371.027,A -85,B 0,C 180,E1 -9610.999,E2 -9610.999} C_VEL
LIN {X 0,Y 431.127,Z 370.341,A -85,B 0,C 180,E1 -9611.957,E2 -9611.957} C_VEL
LIN {X 0,Y 431.23,Z 368.502,A -85,B 0,C 180,E1 -9613.366,E2 -9613.366} C_VEL
LIN {X 0,Y 430.639,Z 367.235,A -85,B 0,C 180,E1 -9614.128,E2 -9614.128} C_VEL
LIN {X 0,Y 427.884,Z 364.593,A -85,B 0,C 180,E1 -9615.354,E2 -9615.354} C_VEL
LIN {X 0,Y 425.594,Z 362.041,A -85,B 0,C 180,E1 -9616.321,E2 -9616.321} C_VEL
LIN {X 0,Y 424.708,Z 359.733,A -85,B 0,C 180,E1 -9617.049,E2 -9617.049} C_VEL
LIN {X 0,Y 424.69,Z 358.88,A -85,B 0,C 180,E1 -9617.29,E2 -9617.29} C_VEL
LIN {X 0,Y 425.028,Z 352.743,A -85,B 0,C 180,E1 -9618.797,E2 -9618.797} C_VEL
LIN {X 0,Y 425.501,Z 345.255,A -85,B 0,C 180,E1 -9620.253,E2 -9620.253} C_VEL
LIN {X 0,Y 425.985,Z 337.629,A -85,B 0,C 180,E1 -9621.461,E2 -9621.461} C_VEL
LIN {X 0,Y 426.608,Z 328.378,A -85,B 0,C 180,E1 -9622.665,E2 -9622.665} C_VEL
LIN {X 0,Y 427.297,Z 318.062,A -85,B 0,C 180,E1 -9623.744,E2 -9623.744} C_VEL
LIN {X 0,Y 427.917,Z 306.643,A -85,B 0,C 180,E1 -9624.699,E2 -9624.699} C_VEL
LIN {X 0,Y 428.511,Z 294.758,A -85,B 0,C 180,E1 -9625.473,E2 -9625.473} C_VEL
LIN {X 0,Y 428.877,Z 282.502,A -85,B 0,C 180,E1 -9626.065,E2 -9626.065} C_VEL
LIN {X 0,Y 429.242,Z 270.298,A -85,B 0,C 180,E1 -9626.469,E2 -9626.469} C_VEL
LIN {X 0,Y 429.485,Z 250.2,A -85,B 0,C 180,E1 -9626.852,E2 -9626.852} C_VEL
LIN {X 0,Y 430.28,Z 179.384,A -85,B 0,C 180,E1 -9628.046,E2 -9628.046} C_VEL
LIN {X 0,Y 426.692,Z 160.753,A -85,B 0,C 180,E1 -9628.52,E2 -9628.52} C_VEL
LIN {X 0,Y 426.802,Z 152.997,A -85,B 0,C 180,E1 -9630.236,E2 -9630.236} C_VEL
LIN {X 0,Y 425.534,Z 145.482,A -85,B 0,C 180,E1 -9632.011,E2 -9632.011} C_VEL
LIN {X 0,Y 425.503,Z 145.483,A -85,B 0,C 180,E1 -9635.688,E2 -9635.688} C_VEL
LIN {X 0,Y 425.39,Z 145.493,A -85,B 0,C 180,E1 -9638.551,E2 -9638.551} C_VEL
LIN {X 0,Y 425.397,Z 145.493,A -85,B 0,C 180,E1 -9642.402,E2 -9642.402} C_VEL
LIN {X 0,Y 425.304,Z 145.504,A -85,B 0,C 180,E1 -9646.315,E2 -9646.315} C_VEL
LIN {X 0,Y 425.288,Z 145.512,A -85,B 0,C 180,E1 -9649.622,E2 -9649.622} C_VEL
LIN {X 0,Y 425.279,Z 145.506,A -85,B 0,C 180,E1 -9652.34,E2 -9652.34} C_VEL
LIN {X 0,Y 425.245,Z 145.518,A -85,B 0,C 180,E1 -9655.449,E2 -9655.449} C_VEL
LIN {X 0,Y 425.292,Z 145.507,A -85,B 0,C 180,E1 -9658.858,E2 -9658.858} C_VEL
LIN {X 0,Y 425.242,Z 145.512,A -85,B 0,C 180,E1 -9661.929,E2 -9661.929} C_VEL
LIN {X 0,Y 425.287,Z 145.511,A -85,B 0,C 180,E1 -9665.338,E2 -9665.338} C_VEL
LIN {X 0,Y 425.271,Z 145.512,A -85,B 0,C 180,E1 -9668.902,E2 -9668.902} C_VEL
LIN {X 0,Y 425.253,Z 145.513,A -85,B 0,C 180,E1 -9672.656,E2 -9672.656} C_VEL
LIN {X 0,Y 425.283,Z 145.509,A -85,B 0,C 180,E1 -9675.284,E2 -9675.284} C_VEL
LIN {X 0,Y 425.246,Z 145.515,A -85,B 0,C 180,E1 -9678.619,E2 -9678.619} C_VEL
LIN {X 0,Y 425.275,Z 145.511,A -85,B 0,C 180,E1 -9681.1,E2 -9681.1} C_VEL
LIN {X 0,Y 425.291,Z 145.512,A -85,B 0,C 180,E1 -9684.664,E2 -9684.664} C_VEL
LIN {X 0,Y 425.246,Z 145.512,A -85,B 0,C 180,E1 -9688.072,E2 -9688.072} C_VEL
LIN {X 0,Y 425.292,Z 145.505,A -85,B 0,C 180,E1 -9691.366,E2 -9691.366} C_VEL
LIN {X 0,Y 425.25,Z 145.516,A -85,B 0,C 180,E1 -9694.552,E2 -9694.552} C_VEL
LIN {X 0,Y 425.291,Z 145.506,A -85,B 0,C 180,E1 -9697.732,E2 -9697.732} C_VEL
LIN {X 0,Y 425.321,Z 145.504,A -85,B 0,C 180,E1 -9700.703,E2 -9700.703} C_VEL
LIN {X 0,Y 425.311,Z 145.504,A -85,B 0,C 180,E1 -9703.686,E2 -9703.686} C_VEL
LIN {X 0,Y 425.405,Z 145.492,A -85,B 0,C 180,E1 -9707.599,E2 -9707.599} C_VEL
LIN {X 0,Y 425.398,Z 145.493,A -85,B 0,C 180,E1 -9711.45,E2 -9711.45} C_VEL
LIN {X 0,Y 425.512,Z 145.481,A -85,B 0,C 180,E1 -9714.313,E2 -9714.313} C_VEL
LIN {X 0,Y 425.568,Z 145.475,A -85,B 0,C 180,E1 -9718.108,E2 -9718.108} C_VEL
LIN {X 0,Y 425.577,Z 145.475,A -85,B 0,C 180,E1 -9720.001,E2 -9720.001} C_VEL
LIN {X 0,Y 425.516,Z 145.477,A -85,B 0,C 180,E1 -9722.841,E2 -9722.841} C_VEL
LIN {X 0,Y 425.477,Z 145.482,A -85,B 0,C 180,E1 -9726.64,E2 -9726.64} C_VEL
LIN {X 0,Y 425.391,Z 145.499,A -85,B 0,C 180,E1 -9729.51,E2 -9729.51} C_VEL
LIN {X 0,Y 425.399,Z 145.493,A -85,B 0,C 180,E1 -9732.904,E2 -9732.904} C_VEL
LIN {X 0,Y 425.323,Z 145.501,A -85,B 0,C 180,E1 -9736.585,E2 -9736.585} C_VEL
LIN {X 0,Y 425.333,Z 145.503,A -85,B 0,C 180,E1 -9739.635,E2 -9739.635} C_VEL
LIN {X 0,Y 425.291,Z 145.505,A -85,B 0,C 180,E1 -9742.339,E2 -9742.339} C_VEL
LIN {X 0,Y 425.263,Z 145.513,A -85,B 0,C 180,E1 -9745.448,E2 -9745.448} C_VEL
LIN {X 0,Y 425.304,Z 145.507,A -85,B 0,C 180,E1 -9748.858,E2 -9748.858} C_VEL
LIN {X 0,Y 425.258,Z 145.509,A -85,B 0,C 180,E1 -9751.928,E2 -9751.928} C_VEL
LIN {X 0,Y 425.299,Z 145.507,A -85,B 0,C 180,E1 -9755.336,E2 -9755.336} C_VEL
LIN {X 0,Y 425.288,Z 145.512,A -85,B 0,C 180,E1 -9758.9,E2 -9758.9} C_VEL
LIN {X 0,Y 425.269,Z 145.508,A -85,B 0,C 180,E1 -9761.954,E2 -9761.954} C_VEL
LIN {X 0,Y 425.289,Z 145.506,A -85,B 0,C 180,E1 -9765.283,E2 -9765.283} C_VEL
LIN {X 0,Y 425.252,Z 145.517,A -85,B 0,C 180,E1 -9768.618,E2 -9768.618} C_VEL
LIN {X 0,Y 425.284,Z 145.507,A -85,B 0,C 180,E1 -9771.099,E2 -9771.099} C_VEL
LIN {X 0,Y 425.299,Z 145.509,A -85,B 0,C 180,E1 -9774.664,E2 -9774.664} C_VEL
LIN {X 0,Y 425.267,Z 145.511,A -85,B 0,C 180,E1 -9778.073,E2 -9778.073} C_VEL
LIN {X 0,Y 425.308,Z 145.506,A -85,B 0,C 180,E1 -9781.366,E2 -9781.366} C_VEL
LIN {X 0,Y 425.365,Z 145.706,A -85,B 0,C 180,E1 -9782.906,E2 -9782.906} C_VEL
LIN {X 0,Y 427.809,Z 158.237,A -85,B 0,C 180,E1 -9785.499,E2 -9785.499} C_VEL
LIN {X 0,Y 427.857,Z 163.521,A -85,B 0,C 180,E1 -9786.526,E2 -9786.526} C_VEL
LIN {X 0,Y 426.777,Z 181.669,A -85,B 0,C 180,E1 -9789.96,E2 -9789.96} C_VEL
LIN {X 0,Y 426.368,Z 189.989,A -85,B 0,C 180,E1 -9791.497,E2 -9791.497} C_VEL
LIN {X 0,Y 429.994,Z 215.321,A -85,B 0,C 180,E1 -9792.075,E2 -9792.075} C_VEL
LIN {X 0,Y 429.106,Z 298.303,A -85,B 0,C 180,E1 -9793.497,E2 -9793.497} C_VEL
LIN {X 0,Y 428.618,Z 311.538,A -85,B 0,C 180,E1 -9793.906,E2 -9793.906} C_VEL
LIN {X 0,Y 428.088,Z 323.715,A -85,B 0,C 180,E1 -9794.466,E2 -9794.466} C_VEL
LIN {X 0,Y 427.454,Z 336.011,A -85,B 0,C 180,E1 -9795.235,E2 -9795.235} C_VEL
LIN {X 0,Y 426.743,Z 347.908,A -85,B 0,C 180,E1 -9796.209,E2 -9796.209} C_VEL
LIN {X 0,Y 426.115,Z 358.118,A -85,B 0,C 180,E1 -9797.256,E2 -9797.256} C_VEL
LIN {X 0,Y 425.617,Z 366.679,A -85,B 0,C 180,E1 -9798.33,E2 -9798.33} C_VEL
LIN {X 0,Y 425.061,Z 374.561,A -85,B 0,C 180,E1 -9799.521,E2 -9799.521} C_VEL
LIN {X 0,Y 424.648,Z 382.256,A -85,B 0,C 180,E1 -9800.954,E2 -9800.954} C_VEL
LIN {X 0,Y 424.371,Z 388.438,A -85,B 0,C 180,E1 -9802.386,E2 -9802.386} C_VEL
LIN {X 0,Y 424.255,Z 392.943,A -85,B 0,C 180,E1 -9803.687,E2 -9803.687} C_VEL
LIN {X 0,Y 424.196,Z 397.101,A -85,B 0,C 180,E1 -9805.248,E2 -9805.248} C_VEL
LIN {X 0,Y 424.101,Z 399.036,A -85,B 0,C 180,E1 -9806.199,E2 -9806.199} C_VEL
LIN {X 0,Y 424.149,Z 400.546,A -85,B 0,C 180,E1 -9807.151,E2 -9807.151} C_VEL
LIN {X 0,Y 424.145,Z 401.599,A -85,B 0,C 180,E1 -9808.101,E2 -9808.101} C_VEL
LIN {X 0,Y 424.112,Z 402.528,A -85,B 0,C 180,E1 -9810,E2 -9810} C_VEL
LIN {X 0,Y 424.094,Z 402.399,A -85,B 0,C 180,E1 -9810.949,E2 -9810.949} C_VEL
LIN {X 0,Y 424.144,Z 401.839,A -85,B 0,C 180,E1 -9811.899,E2 -9811.899} C_VEL
LIN {X 0,Y 424.133,Z 400.885,A -85,B 0,C 180,E1 -9812.849,E2 -9812.849} C_VEL
LIN {X 0,Y 424.099,Z 399.533,A -85,B 0,C 180,E1 -9813.801,E2 -9813.801} C_VEL
LIN {X 0,Y 424.199,Z 396.686,A -85,B 0,C 180,E1 -9815.228,E2 -9815.228} C_VEL
LIN {X 0,Y 424.227,Z 392.811,A -85,B 0,C 180,E1 -9816.659,E2 -9816.659} C_VEL
LIN {X 0,Y 424.505,Z 387.817,A -85,B 0,C 180,E1 -9818.09,E2 -9818.09} C_VEL
LIN {X 0,Y 424.855,Z 381.552,A -85,B 0,C 180,E1 -9819.522,E2 -9819.522} C_VEL
LIN {X 0,Y 425.364,Z 373.741,A -85,B 0,C 180,E1 -9820.953,E2 -9820.953} C_VEL
LIN {X 0,Y 426.15,Z 363.994,A -85,B 0,C 180,E1 -9822.38,E2 -9822.38} C_VEL
LIN {X 0,Y 426.752,Z 354.476,A -85,B 0,C 180,E1 -9823.512,E2 -9823.512} C_VEL
LIN {X 0,Y 427.518,Z 343.972,A -85,B 0,C 180,E1 -9824.519,E2 -9824.519} C_VEL
LIN {X 0,Y 428.368,Z 331.409,A -85,B 0,C 180,E1 -9825.462,E2 -9825.462} C_VEL
LIN {X 0,Y 429.138,Z 319.025,A -85,B 0,C 180,E1 -9826.165,E2 -9826.165} C_VEL
LIN {X 0,Y 429.694,Z 306.788,A -85,B 0,C 180,E1 -9826.663,E2 -9826.663} C_VEL
LIN {X 0,Y 430.198,Z 293.232,A -85,B 0,C 180,E1 -9827.009,E2 -9827.009} C_VEL
LIN {X 0,Y 430.882,Z 214.316,A -85,B 0,C 180,E1 -9828.375,E2 -9828.375} C_VEL
LIN {X 0,Y 427.672,Z 194.304,A -85,B 0,C 180,E1 -9828.895,E2 -9828.895} C_VEL
LIN {X 0,Y 426.783,Z 189.251,A -85,B 0,C 180,E1 -9829.046,E2 -9829.046} C_VEL
LIN {X 0,Y 427.867,Z 171.509,A -85,B 0,C 180,E1 -9832.441,E2 -9832.441} C_VEL
LIN {X 0,Y 428.501,Z 162.391,A -85,B 0,C 180,E1 -9834.207,E2 -9834.207} C_VEL
LIN {X 0,Y 427.557,Z 155.911,A -85,B 0,C 180,E1 -9835.561,E2 -9835.561} C_VEL
LIN {X 0,Y 425.3,Z 145.513,A -85,B 0,C 180,E1 -9837.895,E2 -9837.895} C_VEL
LIN {X 0,Y 425.29,Z 145.513,A -85,B 0,C 180,E1 -9840.816,E2 -9840.816} C_VEL
LIN {X 0,Y 425.293,Z 145.503,A -85,B 0,C 180,E1 -9844.284,E2 -9844.284} C_VEL
LIN {X 0,Y 425.276,Z 145.509,A -85,B 0,C 180,E1 -9847.695,E2 -9847.695} C_VEL
LIN {X 0,Y 425.245,Z 145.51,A -85,B 0,C 180,E1 -9850.514,E2 -9850.514} C_VEL
LIN {X 0,Y 425.248,Z 145.515,A -85,B 0,C 180,E1 -9853.349,E2 -9853.349} C_VEL
LIN {X 0,Y 425.258,Z 145.51,A -85,B 0,C 180,E1 -9856.043,E2 -9856.043} C_VEL
LIN {X 0,Y 425.248,Z 145.515,A -85,B 0,C 180,E1 -9858.618,E2 -9858.618} C_VEL
LIN {X 0,Y 425.275,Z 145.511,A -85,B 0,C 180,E1 -9861.098,E2 -9861.098} C_VEL
LIN {X 0,Y 425.291,Z 145.51,A -85,B 0,C 180,E1 -9864.663,E2 -9864.663} C_VEL
LIN {X 0,Y 425.248,Z 145.512,A -85,B 0,C 180,E1 -9868.071,E2 -9868.071} C_VEL
LIN {X 0,Y 425.294,Z 145.505,A -85,B 0,C 180,E1 -9871.365,E2 -9871.365} C_VEL
LIN {X 0,Y 425.253,Z 145.514,A -85,B 0,C 180,E1 -9874.551,E2 -9874.551} C_VEL
LIN {X 0,Y 425.291,Z 145.499,A -85,B 0,C 180,E1 -9877.73,E2 -9877.73} C_VEL
LIN {X 0,Y 425.321,Z 145.501,A -85,B 0,C 180,E1 -9880.702,E2 -9880.702} C_VEL
LIN {X 0,Y 425.321,Z 145.502,A -85,B 0,C 180,E1 -9883.685,E2 -9883.685} C_VEL
LIN {X 0,Y 425.396,Z 145.485,A -85,B 0,C 180,E1 -9887.097,E2 -9887.097} C_VEL
LIN {X 0,Y 425.389,Z 145.492,A -85,B 0,C 180,E1 -9890.49,E2 -9890.49} C_VEL
LIN {X 0,Y 425.479,Z 145.481,A -85,B 0,C 180,E1 -9893.36,E2 -9893.36} C_VEL
LIN {X 0,Y 425.35,Z 145.499,A -85,B 0,C 180,E1 -9895.261,E2 -9895.261} C_VEL
LIN {X 0,Y 425.567,Z 145.473,A -85,B 0,C 180,E1 -9898.107,E2 -9898.107} C_VEL
LIN {X 0,Y 425.614,Z 145.464,A -85,B 0,C 180,E1 -9899.999,E2 -9899.999} C_VEL
LIN {X 0,Y 425.538,Z 145.473,A -85,B 0,C 180,E1 -9902.839,E2 -9902.839} C_VEL
LIN {X 0,Y 425.482,Z 145.477,A -85,B 0,C 180,E1 -9906.521,E2 -9906.521} C_VEL
LIN {X 0,Y 425.399,Z 145.492,A -85,B 0,C 180,E1 -9909.509,E2 -9909.509} C_VEL
LIN {X 0,Y 425.395,Z 145.497,A -85,B 0,C 180,E1 -9912.903,E2 -9912.903} C_VEL
LIN {X 0,Y 425.362,Z 145.499,A -85,B 0,C 180,E1 -9916.604,E2 -9916.604} C_VEL
LIN {X 0,Y 425.329,Z 145.503,A -85,B 0,C 180,E1 -9919.635,E2 -9919.635} C_VEL
LIN {X 0,Y 425.288,Z 145.504,A -85,B 0,C 180,E1 -9922.338,E2 -9922.338} C_VEL
LIN {X 0,Y 425.32,Z 145.507,A -85,B 0,C 180,E1 -9924.656,E2 -9924.656} C_VEL
LIN {X 0,Y 425.345,Z 145.499,A -85,B 0,C 180,E1 -9927.557,E2 -9927.557} C_VEL
LIN {X 0,Y 425.287,Z 145.51,A -85,B 0,C 180,E1 -9930.815,E2 -9930.815} C_VEL
LIN {X 0,Y 425.309,Z 145.509,A -85,B 0,C 180,E1 -9934.287,E2 -9934.287} C_VEL
LIN {X 0,Y 425.278,Z 145.513,A -85,B 0,C 180,E1 -9937.694,E2 -9937.694} C_VEL
LIN {X 0,Y 425.278,Z 145.518,A -85,B 0,C 180,E1 -9940.52,E2 -9940.52} C_VEL
LIN {X 0,Y 425.256,Z 145.518,A -85,B 0,C 180,E1 -9943.35,E2 -9943.35} C_VEL
LIN {X 0,Y 425.257,Z 145.516,A -85,B 0,C 180,E1 -9946.648,E2 -9946.648} C_VEL
LIN {X 0,Y 425.328,Z 145.62,A -85,B 0,C 180,E1 -9947.411,E2 -9947.411} C_VEL
LIN {X 0,Y 427.211,Z 155.026,A -85,B 0,C 180,E1 -9949.673,E2 -9949.673} C_VEL
LIN {X 0,Y 427.408,Z 159.124,A -85,B 0,C 180,E1 -9950.608,E2 -9950.608} C_VEL
LIN {X 0,Y 427.359,Z 161.207,A -85,B 0,C 180,E1 -9951.046,E2 -9951.046} C_VEL
LIN {X 0,Y 431.506,Z 180.652,A -85,B 0,C 180,E1 -9951.613,E2 -9951.613} C_VEL
LIN {X 0,Y 430.282,Z 268.487,A -85,B 0,C 180,E1 -9953.134,E2 -9953.134} C_VEL
LIN {X 0,Y 429.92,Z 281.122,A -85,B 0,C 180,E1 -9953.532,E2 -9953.532} C_VEL
LIN {X 0,Y 429.422,Z 293.675,A -85,B 0,C 180,E1 -9954.118,E2 -9954.118} C_VEL
LIN {X 0,Y 428.772,Z 305.298,A -85,B 0,C 180,E1 -9954.849,E2 -9954.849} C_VEL
LIN {X 0,Y 428.029,Z 316.682,A -85,B 0,C 180,E1 -9955.78,E2 -9955.78} C_VEL
LIN {X 0,Y 427.258,Z 327.312,A -85,B 0,C 180,E1 -9956.872,E2 -9956.872} C_VEL
LIN {X 0,Y 426.661,Z 335.578,A -85,B 0,C 180,E1 -9957.912,E2 -9957.912} C_VEL
LIN {X 0,Y 425.96,Z 344.271,A -85,B 0,C 180,E1 -9959.238,E2 -9959.238} C_VEL
LIN {X 0,Y 425.359,Z 352.293,A -85,B 0,C 180,E1 -9960.779,E2 -9960.779} C_VEL
LIN {X 0,Y 424.895,Z 358.983,A -85,B 0,C 180,E1 -9962.41,E2 -9962.41} C_VEL
LIN {X 0,Y 424.545,Z 363.888,A -85,B 0,C 180,E1 -9963.98,E2 -9963.98} C_VEL
LIN {X 0,Y 424.283,Z 367.686,A -85,B 0,C 180,E1 -9965.648,E2 -9965.648} C_VEL
LIN {X 0,Y 424.17,Z 369.218,A -85,B 0,C 180,E1 -9966.569,E2 -9966.569} C_VEL
LIN {X 0,Y 424.1,Z 370.927,A -85,B 0,C 180,E1 -9968.125,E2 -9968.125} C_VEL
LIN {X 0,Y 424.031,Z 371.564,A -85,B 0,C 180,E1 -9969.631,E2 -9969.631} C_VEL
LIN {X 0,Y 424.032,Z 371.351,A -85,B 0,C 180,E1 -9970.86,E2 -9970.86} C_VEL
LIN {X 0,Y 424.074,Z 369.855,A -85,B 0,C 180,E1 -9972.644,E2 -9972.644} C_VEL
LIN {X 0,Y 424.234,Z 367.921,A -85,B 0,C 180,E1 -9973.912,E2 -9973.912} C_VEL
LIN {X 0,Y 424.412,Z 364.106,A -85,B 0,C 180,E1 -9975.618,E2 -9975.618} C_VEL
LIN {X 0,Y 424.69,Z 358.88,A -85,B 0,C 180,E1 -9977.29,E2 -9977.29} C_VEL
LIN {X 0,Y 424.229,Z 356.254,A -85,B 0,C 180,E1 -9977.999,E2 -9977.999} C_VEL
LIN {X 0,Y 421.696,Z 351.591,A -85,B 0,C 180,E1 -9979.136,E2 -9979.136} C_VEL
LIN {X 0,Y 419.151,Z 346.338,A -85,B 0,C 180,E1 -9980.233,E2 -9980.233} C_VEL
LIN {X 0,Y 418.677,Z 342.718,A -85,B 0,C 180,E1 -9980.871,E2 -9980.871} C_VEL
LIN {X 0,Y 419.35,Z 333.034,A -85,B 0,C 180,E1 -9982.295,E2 -9982.295} C_VEL
LIN {X 0,Y 419.994,Z 323.763,A -85,B 0,C 180,E1 -9983.394,E2 -9983.394} C_VEL
LIN {X 0,Y 420.734,Z 312.211,A -85,B 0,C 180,E1 -9984.488,E2 -9984.488} C_VEL
LIN {X 0,Y 421.317,Z 300.889,A -85,B 0,C 180,E1 -9985.336,E2 -9985.336} C_VEL
LIN {X 0,Y 421.805,Z 289.376,A -85,B 0,C 180,E1 -9985.999,E2 -9985.999} C_VEL
LIN {X 0,Y 422.172,Z 275.841,A -85,B 0,C 180,E1 -9986.553,E2 -9986.553} C_VEL
LIN {X 0,Y 422.516,Z 262.469,A -85,B 0,C 180,E1 -9986.89,E2 -9986.89} C_VEL
LIN {X 0,Y 423.377,Z 179.757,A -85,B 0,C 180,E1 -9988.31,E2 -9988.31} C_VEL
LIN {X 0,Y 419.779,Z 160.975,A -85,B 0,C 180,E1 -9988.798,E2 -9988.798} C_VEL
LIN {X 0,Y 419.882,Z 154.528,A -85,B 0,C 180,E1 -9990.24,E2 -9990.24} C_VEL
LIN {X 0,Y 418.497,Z 146.359,A -85,B 0,C 180,E1 -9992.196,E2 -9992.196} C_VEL
LIN {X 0,Y 418.464,Z 146.361,A -85,B 0,C 180,E1 -9995.784,E2 -9995.784} C_VEL
LIN {X 0,Y 418.362,Z 146.368,A -85,B 0,C 180,E1 -9998.696,E2 -9998.696} C_VEL
LIN {X 0,Y 418.296,Z 146.382,A -85,B 0,C 180,E1 -10001.632,E2 -10001.632} C_VEL
LIN {X 0,Y 418.272,Z 146.385,A -85,B 0,C 180,E1 -10003.606,E2 -10003.606} C_VEL
LIN {X 0,Y 418.252,Z 146.382,A -85,B 0,C 180,E1 -10006.709,E2 -10006.709} C_VEL
LIN {X 0,Y 418.232,Z 146.389,A -85,B 0,C 180,E1 -10009.777,E2 -10009.777} C_VEL
LIN {X 0,Y 418.218,Z 146.386,A -85,B 0,C 180,E1 -10012.738,E2 -10012.738} C_VEL
LIN {X 0,Y 418.205,Z 146.39,A -85,B 0,C 180,E1 -10015.909,E2 -10015.909} C_VEL
LIN {X 0,Y 418.251,Z 146.387,A -85,B 0,C 180,E1 -10019.163,E2 -10019.163} C_VEL
LIN {X 0,Y 418.227,Z 146.385,A -85,B 0,C 180,E1 -10022.53,E2 -10022.53} C_VEL
LIN {X 0,Y 418.245,Z 146.386,A -85,B 0,C 180,E1 -10024.843,E2 -10024.843} C_VEL
LIN {X 0,Y 418.229,Z 146.385,A -85,B 0,C 180,E1 -10028.445,E2 -10028.445} C_VEL
LIN {X 0,Y 418.215,Z 146.387,A -85,B 0,C 180,E1 -10032.237,E2 -10032.237} C_VEL
LIN {X 0,Y 418.234,Z 146.389,A -85,B 0,C 180,E1 -10035.109,E2 -10035.109} C_VEL
LIN {X 0,Y 418.217,Z 146.386,A -85,B 0,C 180,E1 -10037.765,E2 -10037.765} C_VEL
LIN {X 0,Y 418.233,Z 146.384,A -85,B 0,C 180,E1 -10041.557,E2 -10041.557} C_VEL
LIN {X 0,Y 418.248,Z 146.384,A -85,B 0,C 180,E1 -10045.159,E2 -10045.159} C_VEL
LIN {X 0,Y 418.231,Z 146.385,A -85,B 0,C 180,E1 -10047.471,E2 -10047.471} C_VEL
LIN {X 0,Y 418.258,Z 146.384,A -85,B 0,C 180,E1 -10050.899,E2 -10050.899} C_VEL
LIN {X 0,Y 418.21,Z 146.39,A -85,B 0,C 180,E1 -10054.093,E2 -10054.093} C_VEL
LIN {X 0,Y 418.225,Z 146.385,A -85,B 0,C 180,E1 -10057.264,E2 -10057.264} C_VEL
LIN {X 0,Y 418.248,Z 146.389,A -85,B 0,C 180,E1 -10060.363,E2 -10060.363} C_VEL
LIN {X 0,Y 418.282,Z 146.378,A -85,B 0,C 180,E1 -10063.404,E2 -10063.404} C_VEL
LIN {X 0,Y 418.349,Z 146.37,A -85,B 0,C 180,E1 -10067.386,E2 -10067.386} C_VEL
LIN {X 0,Y 418.324,Z 146.377,A -85,B 0,C 180,E1 -10070.329,E2 -10070.329} C_VEL
LIN {X 0,Y 418.445,Z 146.358,A -85,B 0,C 180,E1 -10073.249,E2 -10073.249} C_VEL
LIN {X 0,Y 418.316,Z 146.374,A -85,B 0,C 180,E1 -10075.182,E2 -10075.182} C_VEL
LIN {X 0,Y 418.537,Z 146.351,A -85,B 0,C 180,E1 -10078.076,E2 -10078.076} C_VEL
LIN {X 0,Y 418.41,Z 146.362,A -85,B 0,C 180,E1 -10080.963,E2 -10080.963} C_VEL
LIN {X 0,Y 418.472,Z 146.354,A -85,B 0,C 180,E1 -10082.888,E2 -10082.888} C_VEL
LIN {X 0,Y 418.443,Z 146.358,A -85,B 0,C 180,E1 -10086.752,E2 -10086.752} C_VEL
LIN {X 0,Y 418.333,Z 146.378,A -85,B 0,C 180,E1 -10089.672,E2 -10089.672} C_VEL
LIN {X 0,Y 418.352,Z 146.371,A -85,B 0,C 180,E1 -10093.001,E2 -10093.001} C_VEL
LIN {X 0,Y 418.269,Z 146.38,A -85,B 0,C 180,E1 -10096.713,E2 -10096.713} C_VEL
LIN {X 0,Y 418.274,Z 146.381,A -85,B 0,C 180,E1 -10099.789,E2 -10099.789} C_VEL
LIN {X 0,Y 418.232,Z 146.386,A -85,B 0,C 180,E1 -10102.737,E2 -10102.737} C_VEL
LIN {X 0,Y 418.223,Z 146.386,A -85,B 0,C 180,E1 -10105.908,E2 -10105.908} C_VEL
LIN {X 0,Y 418.261,Z 146.387,A -85,B 0,C 180,E1 -10109.163,E2 -10109.163} C_VEL
LIN {X 0,Y 418.253,Z 146.387,A -85,B 0,C 180,E1 -10112.842,E2 -10112.842} C_VEL
LIN {X 0,Y 418.248,Z 146.383,A -85,B 0,C 180,E1 -10116.238,E2 -10116.238} C_VEL
LIN {X 0,Y 418.214,Z 146.387,A -85,B 0,C 180,E1 -10119.687,E2 -10119.687} C_VEL
LIN {X 0,Y 418.212,Z 146.389,A -85,B 0,C 180,E1 -10122.318,E2 -10122.318} C_VEL
LIN {X 0,Y 418.24,Z 146.386,A -85,B 0,C 180,E1 -10125.109,E2 -10125.109} C_VEL
LIN {X 0,Y 418.223,Z 146.385,A -85,B 0,C 180,E1 -10127.764,E2 -10127.764} C_VEL
LIN {X 0,Y 418.242,Z 146.383,A -85,B 0,C 180,E1 -10131.556,E2 -10131.556} C_VEL
LIN {X 0,Y 418.254,Z 146.382,A -85,B 0,C 180,E1 -10135.158,E2 -10135.158} C_VEL
LIN {X 0,Y 418.247,Z 146.382,A -85,B 0,C 180,E1 -10137.472,E2 -10137.472} C_VEL
LIN {X 0,Y 418.265,Z 146.385,A -85,B 0,C 180,E1 -10140.897,E2 -10140.897} C_VEL
LIN {X 0,Y 418.28,Z 146.51,A -85,B 0,C 180,E1 -10142.679,E2 -10142.679} C_VEL
LIN {X 0,Y 420.979,Z 160.397,A -85,B 0,C 180,E1 -10145.594,E2 -10145.594} C_VEL
LIN {X 0,Y 420.462,Z 170.974,A -85,B 0,C 180,E1 -10147.65,E2 -10147.65} C_VEL
LIN {X 0,Y 419.367,Z 189.402,A -85,B 0,C 180,E1 -10151.179,E2 -10151.179} C_VEL
LIN {X 0,Y 420.387,Z 196.297,A -85,B 0,C 180,E1 -10151.375,E2 -10151.375} C_VEL
LIN {X 0,Y 423.165,Z 216.895,A -85,B 0,C 180,E1 -10151.844,E2 -10151.844} C_VEL
LIN {X 0,Y 422.254,Z 297.964,A -85,B 0,C 180,E1 -10153.252,E2 -10153.252} C_VEL
LIN {X 0,Y 421.747,Z 311.223,A -85,B 0,C 180,E1 -10153.668,E2 -10153.668} C_VEL
LIN {X 0,Y 421.158,Z 323.981,A -85,B 0,C 180,E1 -10154.266,E2 -10154.266} C_VEL
LIN {X 0,Y 420.533,Z 335.322,A -85,B 0,C 180,E1 -10154.987,E2 -10154.987} C_VEL
LIN {X 0,Y 419.868,Z 346.123,A -85,B 0,C 180,E1 -10155.867,E2 -10155.867} C_VEL
LIN {X 0,Y 419.169,Z 357.572,A -85,B 0,C 180,E1 -10157.041,E2 -10157.041} C_VEL
LIN {X 0,Y 418.628,Z 366.181,A -85,B 0,C 180,E1 -10158.132,E2 -10158.132} C_VEL
LIN {X 0,Y 418.032,Z 374.109,A -85,B 0,C 180,E1 -10159.342,E2 -10159.342} C_VEL
LIN {X 0,Y 417.605,Z 381.848,A -85,B 0,C 180,E1 -10160.8,E2 -10160.8} C_VEL
LIN {X 0,Y 417.322,Z 388.06,A -85,B 0,C 180,E1 -10162.257,E2 -10162.257} C_VEL
LIN {X 0,Y 417.158,Z 393.008,A -85,B 0,C 180,E1 -10163.72,E2 -10163.72} C_VEL
LIN {X 0,Y 417.124,Z 396.773,A -85,B 0,C 180,E1 -10165.167,E2 -10165.167} C_VEL
